LIN {X 0,Y 312.296,Z 514.961,A -85,B 0,C 180,E1 -15750.321,E2 -15750.321} C_VEL
LIN {X 0,Y 313.348,Z 507.271,A -85,B 0,C 180,E1 -15752.248,E2 -15752.248} C_VEL
LIN {X 0,Y 314.368,Z 497.665,A -85,B 0,C 180,E1 -15754.166,E2 -15754.166} C_VEL
LIN {X 0,Y 315.558,Z 488.778,A -85,B 0,C 180,E1 -15755.591,E2 -15755.591} C_VEL
LIN {X 0,Y 316.85,Z 477.877,A -85,B 0,C 180,E1 -15757.006,E2 -15757.006} C_VEL
LIN {X 0,Y 317.928,Z 465.494,A -85,B 0,C 180,E1 -15758.26,E2 -15758.26} C_VEL
LIN {X 0,Y 318.762,Z 453.367,A -85,B 0,C 180,E1 -15759.197,E2 -15759.197} C_VEL
LIN {X 0,Y 319.475,Z 440.605,A -85,B 0,C 180,E1 -15759.895,E2 -15759.895} C_VEL
LIN {X 0,Y 320.059,Z 427.037,A -85,B 0,C 180,E1 -15760.356,E2 -15760.356} C_VEL
LIN {X 0,Y 321.59,Z 354.256,A -85,B 0,C 180,E1 -15761.965,E2 -15761.965} C_VEL
LIN {X 0,Y 318.805,Z 337.841,A -85,B 0,C 180,E1 -15762.528,E2 -15762.528} C_VEL
LIN {X 0,Y 314.195,Z 324.041,A -85,B 0,C 180,E1 -15763.201,E2 -15763.201} C_VEL
LIN {X 0,Y 312.611,Z 316.546,A -85,B 0,C 180,E1 -15765.543,E2 -15765.543} C_VEL
LIN {X 0,Y 312.539,Z 316.555,A -85,B 0,C 180,E1 -15769.711,E2 -15769.711} C_VEL
LIN {X 0,Y 312.518,Z 316.554,A -85,B 0,C 180,E1 -15772.775,E2 -15772.775} C_VEL
LIN {X 0,Y 312.482,Z 316.56,A -85,B 0,C 180,E1 -15776.731,E2 -15776.731} C_VEL
LIN {X 0,Y 312.467,Z 316.56,A -85,B 0,C 180,E1 -15779.657,E2 -15779.657} C_VEL
LIN {X 0,Y 312.518,Z 316.553,A -85,B 0,C 180,E1 -15783.687,E2 -15783.687} C_VEL
LIN {X 0,Y 312.499,Z 316.556,A -85,B 0,C 180,E1 -15787.554,E2 -15787.554} C_VEL
LIN {X 0,Y 311.791,Z 316.649,A -85,B 0,C 180,E1 -15788.629,E2 -15788.629} C_VEL
LIN {X 0,Y 308.92,Z 317.003,A -85,B 0,C 180,E1 -15790.378,E2 -15790.378} C_VEL
LIN {X 0,Y 306.513,Z 317.302,A -85,B 0,C 180,E1 -15791.797,E2 -15791.797} C_VEL
LIN {X 0,Y 305.489,Z 317.434,A -85,B 0,C 180,E1 -15792.895,E2 -15792.895} C_VEL
LIN {X 0,Y 305.409,Z 317.438,A -85,B 0,C 180,E1 -15793.267,E2 -15793.267} C_VEL
LIN {X 0,Y 305.429,Z 317.435,A -85,B 0,C 180,E1 -15797.417,E2 -15797.417} C_VEL
LIN {X 0,Y 305.454,Z 317.434,A -85,B 0,C 180,E1 -15801.594,E2 -15801.594} C_VEL
LIN {X 0,Y 305.455,Z 317.431,A -85,B 0,C 180,E1 -15804.885,E2 -15804.885} C_VEL
LIN {X 0,Y 305.433,Z 317.435,A -85,B 0,C 180,E1 -15808.358,E2 -15808.358} C_VEL
LIN {X 0,Y 305.444,Z 317.437,A -85,B 0,C 180,E1 -15811.105,E2 -15811.105} C_VEL
LIN {X 0,Y 305.471,Z 317.426,A -85,B 0,C 180,E1 -15814.078,E2 -15814.078} C_VEL
LIN {X 0,Y 305.452,Z 317.434,A -85,B 0,C 180,E1 -15818.399,E2 -15818.399} C_VEL
LIN {X 0,Y 305.5,Z 317.428,A -85,B 0,C 180,E1 -15821.212,E2 -15821.212} C_VEL
LIN {X 0,Y 305.558,Z 317.415,A -85,B 0,C 180,E1 -15825.344,E2 -15825.344} C_VEL
LIN {X 0,Y 305.611,Z 317.414,A -85,B 0,C 180,E1 -15829.398,E2 -15829.398} C_VEL
LIN {X 0,Y 305.732,Z 317.402,A -85,B 0,C 180,E1 -15832.072,E2 -15832.072} C_VEL
LIN {X 0,Y 305.652,Z 317.403,A -85,B 0,C 180,E1 -15834.723,E2 -15834.723} C_VEL
LIN {X 0,Y 305.927,Z 317.376,A -85,B 0,C 180,E1 -15838.683,E2 -15838.683} C_VEL
LIN {X 0,Y 305.938,Z 317.372,A -85,B 0,C 180,E1 -15841.316,E2 -15841.316} C_VEL
LIN {X 0,Y 305.79,Z 317.391,A -85,B 0,C 180,E1 -15846.599,E2 -15846.599} C_VEL
LIN {X 0,Y 305.686,Z 317.405,A -85,B 0,C 180,E1 -15849.261,E2 -15849.261} C_VEL
LIN {X 0,Y 305.578,Z 317.417,A -85,B 0,C 180,E1 -15853.296,E2 -15853.296} C_VEL
LIN {X 0,Y 305.544,Z 317.417,A -85,B 0,C 180,E1 -15856.023,E2 -15856.023} C_VEL
LIN {X 0,Y 305.534,Z 317.425,A -85,B 0,C 180,E1 -15859.427,E2 -15859.427} C_VEL
LIN {X 0,Y 305.479,Z 317.433,A -85,B 0,C 180,E1 -15863.04,E2 -15863.04} C_VEL
LIN {X 0,Y 305.497,Z 317.427,A -85,B 0,C 180,E1 -15866.211,E2 -15866.211} C_VEL
LIN {X 0,Y 305.48,Z 317.432,A -85,B 0,C 180,E1 -15869.047,E2 -15869.047} C_VEL
LIN {X 0,Y 305.435,Z 317.435,A -85,B 0,C 180,E1 -15871.953,E2 -15871.953} C_VEL
LIN {X 0,Y 305.455,Z 317.435,A -85,B 0,C 180,E1 -15875.114,E2 -15875.114} C_VEL
LIN {X 0,Y 305.429,Z 317.436,A -85,B 0,C 180,E1 -15878.526,E2 -15878.526} C_VEL
LIN {X 0,Y 305.421,Z 317.438,A -85,B 0,C 180,E1 -15881.86,E2 -15881.86} C_VEL
LIN {X 0,Y 305.395,Z 317.444,A -85,B 0,C 180,E1 -15885.512,E2 -15885.512} C_VEL
LIN {X 0,Y 305.435,Z 317.439,A -85,B 0,C 180,E1 -15888.144,E2 -15888.144} C_VEL
LIN {X 0,Y 305.49,Z 317.432,A -85,B 0,C 180,E1 -15891.601,E2 -15891.601} C_VEL
LIN {X 0,Y 305.459,Z 317.434,A -85,B 0,C 180,E1 -15894.888,E2 -15894.888} C_VEL
LIN {X 0,Y 305.49,Z 317.525,A -85,B 0,C 180,E1 -15898.876,E2 -15898.876} C_VEL
LIN {X 0,Y 307.703,Z 328.091,A -85,B 0,C 180,E1 -15902.083,E2 -15902.083} C_VEL
LIN {X 0,Y 309.104,Z 336.061,A -85,B 0,C 180,E1 -15904.407,E2 -15904.407} C_VEL
LIN {X 0,Y 308.868,Z 340.002,A -85,B 0,C 180,E1 -15905.479,E2 -15905.479} C_VEL
LIN {X 0,Y 313.894,Z 375.423,A -85,B 0,C 180,E1 -15906.683,E2 -15906.683} C_VEL
LIN {X 0,Y 314.544,Z 381.837,A -85,B 0,C 180,E1 -15906.877,E2 -15906.877} C_VEL
LIN {X 0,Y 313.201,Z 448.115,A -85,B 0,C 180,E1 -15908.4,E2 -15908.4} C_VEL
LIN {X 0,Y 312.449,Z 461.495,A -85,B 0,C 180,E1 -15908.951,E2 -15908.951} C_VEL
LIN {X 0,Y 311.441,Z 473.727,A -85,B 0,C 180,E1 -15909.7,E2 -15909.7} C_VEL
LIN {X 0,Y 310.367,Z 485.256,A -85,B 0,C 180,E1 -15910.661,E2 -15910.661} C_VEL
LIN {X 0,Y 309.007,Z 497.067,A -85,B 0,C 180,E1 -15911.949,E2 -15911.949} C_VEL
LIN {X 0,Y 307.847,Z 507.337,A -85,B 0,C 180,E1 -15913.367,E2 -15913.367} C_VEL
LIN {X 0,Y 306.701,Z 517.217,A -85,B 0,C 180,E1 -15915.062,E2 -15915.062} C_VEL
LIN {X 0,Y 305.542,Z 526.379,A -85,B 0,C 180,E1 -15917.041,E2 -15917.041} C_VEL
LIN {X 0,Y 304.7,Z 533.755,A -85,B 0,C 180,E1 -15919.031,E2 -15919.031} C_VEL
LIN {X 0,Y 304.214,Z 538.742,A -85,B 0,C 180,E1 -15920.695,E2 -15920.695} C_VEL
LIN {X 0,Y 303.841,Z 543.574,A -85,B 0,C 180,E1 -15922.692,E2 -15922.692} C_VEL
LIN {X 0,Y 303.637,Z 547.267,A -85,B 0,C 180,E1 -15924.689,E2 -15924.689} C_VEL
LIN {X 0,Y 303.637,Z 549.173,A -85,B 0,C 180,E1 -15926.019,E2 -15926.019} C_VEL
LIN {X 0,Y 303.614,Z 550.618,A -85,B 0,C 180,E1 -15927.348,E2 -15927.348} C_VEL
LIN {X 0,Y 303.579,Z 551.634,A -85,B 0,C 180,E1 -15928.674,E2 -15928.674} C_VEL
LIN {X 0,Y 303.605,Z 552.26,A -85,B 0,C 180,E1 -15930.001,E2 -15930.001} C_VEL
LIN {X 0,Y 303.573,Z 552.497,A -85,B 0,C 180,E1 -15931.328,E2 -15931.328} C_VEL
LIN {X 0,Y 303.601,Z 552.318,A -85,B 0,C 180,E1 -15932.655,E2 -15932.655} C_VEL
LIN {X 0,Y 303.638,Z 550.75,A -85,B 0,C 180,E1 -15935.313,E2 -15935.313} C_VEL
LIN {X 0,Y 303.755,Z 549.383,A -85,B 0,C 180,E1 -15936.644,E2 -15936.644} C_VEL
LIN {X 0,Y 304.19,Z 546.513,A -85,B 0,C 180,E1 -15938.638,E2 -15938.638} C_VEL
LIN {X 0,Y 304.838,Z 542.633,A -85,B 0,C 180,E1 -15940.629,E2 -15940.629} C_VEL
LIN {X 0,Y 305.776,Z 537.648,A -85,B 0,C 180,E1 -15942.613,E2 -15942.613} C_VEL
LIN {X 0,Y 307.136,Z 531.405,A -85,B 0,C 180,E1 -15944.579,E2 -15944.579} C_VEL
LIN {X 0,Y 308.798,Z 523.623,A -85,B 0,C 180,E1 -15946.529,E2 -15946.529} C_VEL
LIN {X 0,Y 310.409,Z 514.991,A -85,B 0,C 180,E1 -15948.278,E2 -15948.278} C_VEL
LIN {X 0,Y 312.375,Z 505.012,A -85,B 0,C 180,E1 -15949.895,E2 -15949.895} C_VEL
LIN {X 0,Y 314.343,Z 494.038,A -85,B 0,C 180,E1 -15951.305,E2 -15951.305} C_VEL
LIN {X 0,Y 316.047,Z 483.306,A -85,B 0,C 180,E1 -15952.385,E2 -15952.385} C_VEL
LIN {X 0,Y 317.554,Z 471.518,A -85,B 0,C 180,E1 -15953.304,E2 -15953.304} C_VEL
LIN {X 0,Y 318.911,Z 458.823,A -85,B 0,C 180,E1 -15954.018,E2 -15954.018} C_VEL
LIN {X 0,Y 319.693,Z 446.646,A -85,B 0,C 180,E1 -15954.473,E2 -15954.473} C_VEL
LIN {X 0,Y 321.429,Z 382.108,A -85,B 0,C 180,E1 -15955.952,E2 -15955.952} C_VEL
LIN {X 0,Y 317.863,Z 362.317,A -85,B 0,C 180,E1 -15956.829,E2 -15956.829} C_VEL
LIN {X 0,Y 315.108,Z 349.801,A -85,B 0,C 180,E1 -15957.454,E2 -15957.454} C_VEL
LIN {X 0,Y 310.693,Z 339.327,A -85,B 0,C 180,E1 -15958.249,E2 -15958.249} C_VEL
LIN {X 0,Y 308.404,Z 329.1,A -85,B 0,C 180,E1 -15961.611,E2 -15961.611} C_VEL
LIN {X 0,Y 305.969,Z 319.3,A -85,B 0,C 180,E1 -15965.047,E2 -15965.047} C_VEL
LIN {X 0,Y 305.494,Z 317.433,A -85,B 0,C 180,E1 -15965.818,E2 -15965.818} C_VEL
LIN {X 0,Y 305.459,Z 317.436,A -85,B 0,C 180,E1 -15970.108,E2 -15970.108} C_VEL
LIN {X 0,Y 305.427,Z 317.437,A -85,B 0,C 180,E1 -15973.656,E2 -15973.656} C_VEL
LIN {X 0,Y 305.456,Z 317.436,A -85,B 0,C 180,E1 -15977.415,E2 -15977.415} C_VEL
LIN {X 0,Y 305.459,Z 317.434,A -85,B 0,C 180,E1 -15979.893,E2 -15979.893} C_VEL
LIN {X 0,Y 305.465,Z 317.433,A -85,B 0,C 180,E1 -15983.637,E2 -15983.637} C_VEL
LIN {X 0,Y 305.467,Z 317.435,A -85,B 0,C 180,E1 -15986.484,E2 -15986.484} C_VEL
LIN {X 0,Y 305.437,Z 317.438,A -85,B 0,C 180,E1 -15989.588,E2 -15989.588} C_VEL
LIN {X 0,Y 305.473,Z 317.43,A -85,B 0,C 180,E1 -15992.604,E2 -15992.604} C_VEL
LIN {X 0,Y 305.49,Z 317.426,A -85,B 0,C 180,E1 -15995.537,E2 -15995.537} C_VEL
LIN {X 0,Y 305.486,Z 317.428,A -85,B 0,C 180,E1 -15999.813,E2 -15999.813} C_VEL
LIN {X 0,Y 305.556,Z 317.418,A -85,B 0,C 180,E1 -16003.978,E2 -16003.978} C_VEL
LIN {X 0,Y 305.588,Z 317.412,A -85,B 0,C 180,E1 -16006.704,E2 -16006.704} C_VEL
LIN {X 0,Y 305.758,Z 317.389,A -85,B 0,C 180,E1 -16011.258,E2 -16011.258} C_VEL
LIN {X 0,Y 305.833,Z 317.382,A -85,B 0,C 180,E1 -16013.402,E2 -16013.402} C_VEL
LIN {X 0,Y 305.951,Z 317.368,A -85,B 0,C 180,E1 -16018.684,E2 -16018.684} C_VEL
LIN {X 0,Y 305.952,Z 317.364,A -85,B 0,C 180,E1 -16021.317,E2 -16021.317} C_VEL
LIN {X 0,Y 305.672,Z 317.399,A -85,B 0,C 180,E1 -16025.277,E2 -16025.277} C_VEL
LIN {X 0,Y 305.767,Z 317.396,A -85,B 0,C 180,E1 -16027.927,E2 -16027.927} C_VEL
LIN {X 0,Y 305.602,Z 317.417,A -85,B 0,C 180,E1 -16031.945,E2 -16031.945} C_VEL
LIN {X 0,Y 305.612,Z 317.418,A -85,B 0,C 180,E1 -16035.015,E2 -16035.015} C_VEL
LIN {X 0,Y 305.547,Z 317.423,A -85,B 0,C 180,E1 -16039.427,E2 -16039.427} C_VEL
LIN {X 0,Y 305.489,Z 317.431,A -85,B 0,C 180,E1 -16043.039,E2 -16043.039} C_VEL
LIN {X 0,Y 305.481,Z 317.428,A -85,B 0,C 180,E1 -16046.2,E2 -16046.2} C_VEL
LIN {X 0,Y 305.466,Z 317.428,A -85,B 0,C 180,E1 -16049.039,E2 -16049.039} C_VEL
LIN {X 0,Y 305.44,Z 317.432,A -85,B 0,C 180,E1 -16051.953,E2 -16051.953} C_VEL
LIN {X 0,Y 305.466,Z 317.43,A -85,B 0,C 180,E1 -16055.113,E2 -16055.113} C_VEL
LIN {X 0,Y 305.452,Z 317.437,A -85,B 0,C 180,E1 -16058.528,E2 -16058.528} C_VEL
LIN {X 0,Y 305.458,Z 317.436,A -85,B 0,C 180,E1 -16062.586,E2 -16062.586} C_VEL
LIN {X 0,Y 305.425,Z 317.441,A -85,B 0,C 180,E1 -16066.344,E2 -16066.344} C_VEL
LIN {X 0,Y 305.439,Z 317.538,A -85,B 0,C 180,E1 -16067.751,E2 -16067.751} C_VEL
LIN {X 0,Y 307.326,Z 324.783,A -85,B 0,C 180,E1 -16070.4,E2 -16070.4} C_VEL
LIN {X 0,Y 316.814,Z 344.367,A -85,B 0,C 180,E1 -16072.019,E2 -16072.019} C_VEL
LIN {X 0,Y 321.176,Z 354.703,A -85,B 0,C 180,E1 -16072.753,E2 -16072.753} C_VEL
LIN {X 0,Y 322.117,Z 358.964,A -85,B 0,C 180,E1 -16072.96,E2 -16072.96} C_VEL
LIN {X 0,Y 319.954,Z 432.294,A -85,B 0,C 180,E1 -16074.634,E2 -16074.634} C_VEL
LIN {X 0,Y 319.069,Z 445.156,A -85,B 0,C 180,E1 -16075.157,E2 -16075.157} C_VEL
LIN {X 0,Y 317.781,Z 458.257,A -85,B 0,C 180,E1 -16075.957,E2 -16075.957} C_VEL
LIN {X 0,Y 316.528,Z 468.963,A -85,B 0,C 180,E1 -16076.854,E2 -16076.854} C_VEL
LIN {X 0,Y 314.836,Z 480.903,A -85,B 0,C 180,E1 -16078.156,E2 -16078.156} C_VEL
LIN {X 0,Y 312.867,Z 491.723,A -85,B 0,C 180,E1 -16079.64,E2 -16079.64} C_VEL
LIN {X 0,Y 310.97,Z 501.278,A -85,B 0,C 180,E1 -16081.297,E2 -16081.297} C_VEL
LIN {X 0,Y 309.069,Z 510.472,A -85,B 0,C 180,E1 -16083.313,E2 -16083.313} C_VEL
LIN {X 0,Y 307.444,Z 517.806,A -85,B 0,C 180,E1 -16085.342,E2 -16085.342} C_VEL
LIN {X 0,Y 306.397,Z 522.72,A -85,B 0,C 180,E1 -16087.049,E2 -16087.049} C_VEL
LIN {X 0,Y 305.343,Z 527.44,A -85,B 0,C 180,E1 -16089.098,E2 -16089.098} C_VEL
LIN {X 0,Y 304.609,Z 530.992,A -85,B 0,C 180,E1 -16091.154,E2 -16091.154} C_VEL
LIN {X 0,Y 304.184,Z 532.749,A -85,B 0,C 180,E1 -16092.52,E2 -16092.52} C_VEL
LIN {X 0,Y 303.878,Z 534.072,A -85,B 0,C 180,E1 -16093.886,E2 -16093.886} C_VEL
LIN {X 0,Y 303.634,Z 535.444,A -85,B 0,C 180,E1 -16096.447,E2 -16096.447} C_VEL
LIN {X 0,Y 303.5,Z 535.534,A -85,B 0,C 180,E1 -16097.97,E2 -16097.97} C_VEL
LIN {X 0,Y 303.445,Z 534.477,A -85,B 0,C 180,E1 -16100.669,E2 -16100.669} C_VEL
LIN {X 0,Y 303.521,Z 533.321,A -85,B 0,C 180,E1 -16102.013,E2 -16102.013} C_VEL
LIN {X 0,Y 303.798,Z 530.629,A -85,B 0,C 180,E1 -16104.134,E2 -16104.134} C_VEL
LIN {X 0,Y 304.077,Z 527.294,A -85,B 0,C 180,E1 -16106.023,E2 -16106.023} C_VEL
LIN {X 0,Y 304.507,Z 522.685,A -85,B 0,C 180,E1 -16108.015,E2 -16108.015} C_VEL
LIN {X 0,Y 305.18,Z 515.732,A -85,B 0,C 180,E1 -16110.329,E2 -16110.329} C_VEL
LIN {X 0,Y 306.278,Z 508.187,A -85,B 0,C 180,E1 -16112.3,E2 -16112.3} C_VEL
LIN {X 0,Y 307.123,Z 500.516,A -85,B 0,C 180,E1 -16113.935,E2 -16113.935} C_VEL
LIN {X 0,Y 308.265,Z 491.148,A -85,B 0,C 180,E1 -16115.559,E2 -16115.559} C_VEL
LIN {X 0,Y 309.678,Z 480.703,A -85,B 0,C 180,E1 -16117.006,E2 -16117.006} C_VEL
LIN {X 0,Y 310.816,Z 469.157,A -85,B 0,C 180,E1 -16118.287,E2 -16118.287} C_VEL
LIN {X 0,Y 311.744,Z 456.945,A -85,B 0,C 180,E1 -16119.324,E2 -16119.324} C_VEL
LIN {X 0,Y 312.536,Z 444.098,A -85,B 0,C 180,E1 -16120.117,E2 -16120.117} C_VEL
LIN {X 0,Y 313.129,Z 431.64,A -85,B 0,C 180,E1 -16120.629,E2 -16120.629} C_VEL
LIN {X 0,Y 314.902,Z 355.1,A -85,B 0,C 180,E1 -16122.373,E2 -16122.373} C_VEL
LIN {X 0,Y 312.167,Z 339.4,A -85,B 0,C 180,E1 -16122.932,E2 -16122.932} C_VEL
LIN {X 0,Y 307.042,Z 324.32,A -85,B 0,C 180,E1 -16123.673,E2 -16123.673} C_VEL
LIN {X 0,Y 305.557,Z 317.426,A -85,B 0,C 180,E1 -16125.894,E2 -16125.894} C_VEL
LIN {X 0,Y 305.484,Z 317.435,A -85,B 0,C 180,E1 -16130.186,E2 -16130.186} C_VEL
LIN {X 0,Y 305.456,Z 317.437,A -85,B 0,C 180,E1 -16134.464,E2 -16134.464} C_VEL
LIN {X 0,Y 305.441,Z 317.435,A -85,B 0,C 180,E1 -16137.398,E2 -16137.398} C_VEL
LIN {X 0,Y 305.415,Z 317.442,A -85,B 0,C 180,E1 -16140.413,E2 -16140.413} C_VEL
LIN {X 0,Y 305.463,Z 317.433,A -85,B 0,C 180,E1 -16144.077,E2 -16144.077} C_VEL
LIN {X 0,Y 305.429,Z 317.436,A -85,B 0,C 180,E1 -16147.552,E2 -16147.552} C_VEL
LIN {X 0,Y 305.407,Z 317.438,A -85,B 0,C 180,E1 -16151.861,E2 -16151.861} C_VEL
LIN {X 0,Y 305.409,Z 317.438,A -85,B 0,C 180,E1 -16153.267,E2 -16153.267} C_VEL
LIN {X 0,Y 304.752,Z 317.523,A -85,B 0,C 180,E1 -16154.368,E2 -16154.368} C_VEL
LIN {X 0,Y 301.911,Z 317.881,A -85,B 0,C 180,E1 -16156.161,E2 -16156.161} C_VEL
LIN {X 0,Y 299.484,Z 318.183,A -85,B 0,C 180,E1 -16157.615,E2 -16157.615} C_VEL
LIN {X 0,Y 298.428,Z 318.311,A -85,B 0,C 180,E1 -16158.74,E2 -16158.74} C_VEL
LIN {X 0,Y 298.333,Z 318.32,A -85,B 0,C 180,E1 -16159.122,E2 -16159.122} C_VEL
LIN {X 0,Y 298.422,Z 318.31,A -85,B 0,C 180,E1 -16163.196,E2 -16163.196} C_VEL
LIN {X 0,Y 298.402,Z 318.31,A -85,B 0,C 180,E1 -16165.58,E2 -16165.58} C_VEL
LIN {X 0,Y 298.363,Z 318.317,A -85,B 0,C 180,E1 -16168.787,E2 -16168.787} C_VEL
LIN {X 0,Y 298.387,Z 318.312,A -85,B 0,C 180,E1 -16171.896,E2 -16171.896} C_VEL
LIN {X 0,Y 298.414,Z 318.304,A -85,B 0,C 180,E1 -16174.917,E2 -16174.917} C_VEL
LIN {X 0,Y 298.408,Z 318.313,A -85,B 0,C 180,E1 -16179.312,E2 -16179.312} C_VEL
LIN {X 0,Y 298.43,Z 318.307,A -85,B 0,C 180,E1 -16182.172,E2 -16182.172} C_VEL
LIN {X 0,Y 298.502,Z 318.291,A -85,B 0,C 180,E1 -16184.99,E2 -16184.99} C_VEL
LIN {X 0,Y 298.569,Z 318.29,A -85,B 0,C 180,E1 -16189.145,E2 -16189.145} C_VEL
LIN {X 0,Y 298.677,Z 318.281,A -85,B 0,C 180,E1 -16191.883,E2 -16191.883} C_VEL
LIN {X 0,Y 298.622,Z 318.278,A -85,B 0,C 180,E1 -16194.598,E2 -16194.598} C_VEL
LIN {X 0,Y 298.895,Z 318.252,A -85,B 0,C 180,E1 -16198.652,E2 -16198.652} C_VEL
LIN {X 0,Y 298.905,Z 318.249,A -85,B 0,C 180,E1 -16201.347,E2 -16201.347} C_VEL
LIN {X 0,Y 298.739,Z 318.27,A -85,B 0,C 180,E1 -16206.755,E2 -16206.755} C_VEL
LIN {X 0,Y 298.617,Z 318.284,A -85,B 0,C 180,E1 -16209.482,E2 -16209.482} C_VEL
LIN {X 0,Y 298.537,Z 318.292,A -85,B 0,C 180,E1 -16213.616,E2 -16213.616} C_VEL
LIN {X 0,Y 298.478,Z 318.298,A -85,B 0,C 180,E1 -16216.412,E2 -16216.412} C_VEL
LIN {X 0,Y 298.475,Z 318.303,A -85,B 0,C 180,E1 -16219.639,E2 -16219.639} C_VEL
LIN {X 0,Y 298.418,Z 318.31,A -85,B 0,C 180,E1 -16223.601,E2 -16223.601} C_VEL
LIN {X 0,Y 298.448,Z 318.307,A -85,B 0,C 180,E1 -16226.578,E2 -16226.578} C_VEL
LIN {X 0,Y 298.409,Z 318.313,A -85,B 0,C 180,E1 -16229.642,E2 -16229.642} C_VEL
LIN {X 0,Y 298.388,Z 318.313,A -85,B 0,C 180,E1 -16232.801,E2 -16232.801} C_VEL
LIN {X 0,Y 298.422,Z 318.309,A -85,B 0,C 180,E1 -16236.804,E2 -16236.804} C_VEL
LIN {X 0,Y 298.375,Z 318.315,A -85,B 0,C 180,E1 -16241.087,E2 -16241.087} C_VEL
LIN {X 0,Y 298.393,Z 318.311,A -85,B 0,C 180,E1 -16243.104,E2 -16243.104} C_VEL
LIN {X 0,Y 298.398,Z 318.312,A -85,B 0,C 180,E1 -16246.922,E2 -16246.922} C_VEL
LIN {X 0,Y 298.41,Z 318.311,A -85,B 0,C 180,E1 -16251.005,E2 -16251.005} C_VEL
LIN {X 0,Y 298.415,Z 318.315,A -85,B 0,C 180,E1 -16253.931,E2 -16253.931} C_VEL
LIN {X 0,Y 298.394,Z 318.319,A -85,B 0,C 180,E1 -16257.984,E2 -16257.984} C_VEL
LIN {X 0,Y 298.443,Z 318.417,A -85,B 0,C 180,E1 -16258.511,E2 -16258.511} C_VEL
LIN {X 0,Y 300.623,Z 328.791,A -85,B 0,C 180,E1 -16261.746,E2 -16261.746} C_VEL
LIN {X 0,Y 302.175,Z 338.091,A -85,B 0,C 180,E1 -16264.516,E2 -16264.516} C_VEL
LIN {X 0,Y 302.038,Z 339.794,A -85,B 0,C 180,E1 -16264.987,E2 -16264.987} C_VEL
LIN {X 0,Y 306.832,Z 373.458,A -85,B 0,C 180,E1 -16266.173,E2 -16266.173} C_VEL
LIN {X 0,Y 307.838,Z 382.335,A -85,B 0,C 180,E1 -16266.457,E2 -16266.457} C_VEL
LIN {X 0,Y 306.415,Z 448.885,A -85,B 0,C 180,E1 -16268.03,E2 -16268.03} C_VEL
LIN {X 0,Y 305.573,Z 462.705,A -85,B 0,C 180,E1 -16268.631,E2 -16268.631} C_VEL
LIN {X 0,Y 304.504,Z 475.613,A -85,B 0,C 180,E1 -16269.482,E2 -16269.482} C_VEL
LIN {X 0,Y 303.319,Z 487.411,A -85,B 0,C 180,E1 -16270.546,E2 -16270.546} C_VEL
LIN {X 0,Y 301.871,Z 498.77,A -85,B 0,C 180,E1 -16271.858,E2 -16271.858} C_VEL
LIN {X 0,Y 300.694,Z 509.168,A -85,B 0,C 180,E1 -16273.391,E2 -16273.391} C_VEL
LIN {X 0,Y 299.553,Z 518.223,A -85,B 0,C 180,E1 -16275.045,E2 -16275.045} C_VEL
LIN {X 0,Y 298.409,Z 527.186,A -85,B 0,C 180,E1 -16277.072,E2 -16277.072} C_VEL
LIN {X 0,Y 297.576,Z 534.367,A -85,B 0,C 180,E1 -16279.11,E2 -16279.11} C_VEL
LIN {X 0,Y 297.014,Z 540.079,A -85,B 0,C 180,E1 -16281.154,E2 -16281.154} C_VEL
LIN {X 0,Y 296.693,Z 544.567,A -85,B 0,C 180,E1 -16283.199,E2 -16283.199} C_VEL
LIN {X 0,Y 296.551,Z 546.928,A -85,B 0,C 180,E1 -16284.561,E2 -16284.561} C_VEL
LIN {X 0,Y 296.534,Z 548.857,A -85,B 0,C 180,E1 -16285.924,E2 -16285.924} C_VEL
LIN {X 0,Y 296.54,Z 550.346,A -85,B 0,C 180,E1 -16287.284,E2 -16287.284} C_VEL
LIN {X 0,Y 296.498,Z 551.383,A -85,B 0,C 180,E1 -16288.643,E2 -16288.643} C_VEL
LIN {X 0,Y 296.52,Z 552.03,A -85,B 0,C 180,E1 -16290.001,E2 -16290.001} C_VEL
LIN {X 0,Y 296.492,Z 552.288,A -85,B 0,C 180,E1 -16291.359,E2 -16291.359} C_VEL
LIN {X 0,Y 296.526,Z 552.148,A -85,B 0,C 180,E1 -16292.718,E2 -16292.718} C_VEL
LIN {X 0,Y 296.554,Z 550.625,A -85,B 0,C 180,E1 -16295.44,E2 -16295.44} C_VEL
LIN {X 0,Y 296.699,Z 549.281,A -85,B 0,C 180,E1 -16296.803,E2 -16296.803} C_VEL
LIN {X 0,Y 297.163,Z 546.456,A -85,B 0,C 180,E1 -16298.844,E2 -16298.844} C_VEL
LIN {X 0,Y 297.833,Z 542.625,A -85,B 0,C 180,E1 -16300.882,E2 -16300.882} C_VEL
LIN {X 0,Y 298.836,Z 537.691,A -85,B 0,C 180,E1 -16302.911,E2 -16302.911} C_VEL
LIN {X 0,Y 300.271,Z 531.505,A -85,B 0,C 180,E1 -16304.92,E2 -16304.92} C_VEL
LIN {X 0,Y 301.981,Z 523.823,A -85,B 0,C 180,E1 -16306.913,E2 -16306.913} C_VEL
LIN {X 0,Y 303.883,Z 514.218,A -85,B 0,C 180,E1 -16308.893,E2 -16308.893} C_VEL
LIN {X 0,Y 305.964,Z 504.32,A -85,B 0,C 180,E1 -16310.506,E2 -16310.506} C_VEL
LIN {X 0,Y 308.055,Z 493.18,A -85,B 0,C 180,E1 -16311.937,E2 -16311.937} C_VEL
LIN {X 0,Y 309.787,Z 482.295,A -85,B 0,C 180,E1 -16313.039,E2 -16313.039} C_VEL
LIN {X 0,Y 311.382,Z 470.284,A -85,B 0,C 180,E1 -16313.971,E2 -16313.971} C_VEL
LIN {X 0,Y 312.662,Z 457.946,A -85,B 0,C 180,E1 -16314.662,E2 -16314.662} C_VEL
LIN {X 0,Y 313.538,Z 445.216,A -85,B 0,C 180,E1 -16315.119,E2 -16315.119} C_VEL
LIN {X 0,Y 315.256,Z 383.061,A -85,B 0,C 180,E1 -16316.568,E2 -16316.568} C_VEL
LIN {X 0,Y 311.286,Z 361.291,A -85,B 0,C 180,E1 -16317.575,E2 -16317.575} C_VEL
LIN {X 0,Y 309.205,Z 352.32,A -85,B 0,C 180,E1 -16318.052,E2 -16318.052} C_VEL
LIN {X 0,Y 304.326,Z 341.341,A -85,B 0,C 180,E1 -16318.928,E2 -16318.928} C_VEL
LIN {X 0,Y 303.478,Z 339.127,A -85,B 0,C 180,E1 -16319.1,E2 -16319.1} C_VEL
LIN {X 0,Y 300.994,Z 328.318,A -85,B 0,C 180,E1 -16322.799,E2 -16322.799} C_VEL
LIN {X 0,Y 298.449,Z 318.312,A -85,B 0,C 180,E1 -16326.49,E2 -16326.49} C_VEL
LIN {X 0,Y 298.401,Z 318.313,A -85,B 0,C 180,E1 -16329.488,E2 -16329.488} C_VEL
LIN {X 0,Y 298.401,Z 318.314,A -85,B 0,C 180,E1 -16333.104,E2 -16333.104} C_VEL
LIN {X 0,Y 298.405,Z 318.315,A -85,B 0,C 180,E1 -16336.921,E2 -16336.921} C_VEL
LIN {X 0,Y 298.392,Z 318.311,A -85,B 0,C 180,E1 -16341.01,E2 -16341.01} C_VEL
LIN {X 0,Y 298.407,Z 318.312,A -85,B 0,C 180,E1 -16343.929,E2 -16343.929} C_VEL
LIN {X 0,Y 298.395,Z 318.311,A -85,B 0,C 180,E1 -16347.2,E2 -16347.2} C_VEL
LIN {X 0,Y 298.412,Z 318.311,A -85,B 0,C 180,E1 -16350.622,E2 -16350.622} C_VEL
LIN {X 0,Y 298.452,Z 318.303,A -85,B 0,C 180,E1 -16354.921,E2 -16354.921} C_VEL
LIN {X 0,Y 298.416,Z 318.31,A -85,B 0,C 180,E1 -16357.864,E2 -16357.864} C_VEL
LIN {X 0,Y 298.48,Z 318.302,A -85,B 0,C 180,E1 -16360.753,E2 -16360.753} C_VEL
LIN {X 0,Y 298.588,Z 318.288,A -85,B 0,C 180,E1 -16364.995,E2 -16364.995} C_VEL
LIN {X 0,Y 298.593,Z 318.285,A -85,B 0,C 180,E1 -16369.147,E2 -16369.147} C_VEL
LIN {X 0,Y 298.719,Z 318.264,A -85,B 0,C 180,E1 -16371.885,E2 -16371.885} C_VEL
LIN {X 0,Y 298.649,Z 318.276,A -85,B 0,C 180,E1 -16374.599,E2 -16374.599} C_VEL
LIN {X 0,Y 298.918,Z 318.244,A -85,B 0,C 180,E1 -16378.653,E2 -16378.653} C_VEL
LIN {X 0,Y 298.919,Z 318.24,A -85,B 0,C 180,E1 -16381.347,E2 -16381.347} C_VEL
LIN {X 0,Y 298.748,Z 318.27,A -85,B 0,C 180,E1 -16386.755,E2 -16386.755} C_VEL
LIN {X 0,Y 298.628,Z 318.276,A -85,B 0,C 180,E1 -16389.482,E2 -16389.482} C_VEL
LIN {X 0,Y 298.548,Z 318.287,A -85,B 0,C 180,E1 -16393.616,E2 -16393.616} C_VEL
LIN {X 0,Y 298.49,Z 318.302,A -85,B 0,C 180,E1 -16396.412,E2 -16396.412} C_VEL
LIN {X 0,Y 298.487,Z 318.302,A -85,B 0,C 180,E1 -16399.64,E2 -16399.64} C_VEL
LIN {X 0,Y 298.427,Z 318.308,A -85,B 0,C 180,E1 -16403.601,E2 -16403.601} C_VEL
LIN {X 0,Y 298.42,Z 318.309,A -85,B 0,C 180,E1 -16406.582,E2 -16406.582} C_VEL
LIN {X 0,Y 298.403,Z 318.313,A -85,B 0,C 180,E1 -16409.643,E2 -16409.643} C_VEL
LIN {X 0,Y 298.396,Z 318.313,A -85,B 0,C 180,E1 -16412.801,E2 -16412.801} C_VEL
LIN {X 0,Y 298.45,Z 318.307,A -85,B 0,C 180,E1 -16416.808,E2 -16416.808} C_VEL
LIN {X 0,Y 298.391,Z 318.318,A -85,B 0,C 180,E1 -16421.088,E2 -16421.088} C_VEL
LIN {X 0,Y 298.403,Z 318.316,A -85,B 0,C 180,E1 -16423.103,E2 -16423.103} C_VEL
LIN {X 0,Y 298.395,Z 318.392,A -85,B 0,C 180,E1 -16426.998,E2 -16426.998} C_VEL
LIN {X 0,Y 300.211,Z 325.283,A -85,B 0,C 180,E1 -16429.537,E2 -16429.537} C_VEL
LIN {X 0,Y 308.112,Z 340.972,A -85,B 0,C 180,E1 -16430.942,E2 -16430.942} C_VEL
LIN {X 0,Y 315.261,Z 357.011,A -85,B 0,C 180,E1 -16432.179,E2 -16432.179} C_VEL
LIN {X 0,Y 316.009,Z 361.29,A -85,B 0,C 180,E1 -16432.373,E2 -16432.373} C_VEL
LIN {X 0,Y 313.693,Z 433.005,A -85,B 0,C 180,E1 -16434.037,E2 -16434.037} C_VEL
LIN {X 0,Y 312.808,Z 445.372,A -85,B 0,C 180,E1 -16434.553,E2 -16434.553} C_VEL
LIN {X 0,Y 311.474,Z 458.463,A -85,B 0,C 180,E1 -16435.366,E2 -16435.366} C_VEL
LIN {X 0,Y 310.168,Z 469.162,A -85,B 0,C 180,E1 -16436.279,E2 -16436.279} C_VEL
LIN {X 0,Y 308.668,Z 479.473,A -85,B 0,C 180,E1 -16437.4,E2 -16437.4} C_VEL
LIN {X 0,Y 306.558,Z 490.814,A -85,B 0,C 180,E1 -16438.947,E2 -16438.947} C_VEL
LIN {X 0,Y 304.555,Z 500.621,A -85,B 0,C 180,E1 -16440.634,E2 -16440.634} C_VEL
LIN {X 0,Y 302.827,Z 508.579,A -85,B 0,C 180,E1 -16442.343,E2 -16442.343} C_VEL
LIN {X 0,Y 301.056,Z 516.298,A -85,B 0,C 180,E1 -16444.413,E2 -16444.413} C_VEL
LIN {X 0,Y 299.607,Z 522.452,A -85,B 0,C 180,E1 -16446.498,E2 -16446.498} C_VEL
LIN {X 0,Y 298.464,Z 527.274,A -85,B 0,C 180,E1 -16448.593,E2 -16448.593} C_VEL
LIN {X 0,Y 297.6,Z 531.15,A -85,B 0,C 180,E1 -16450.845,E2 -16450.845} C_VEL
LIN {X 0,Y 297.213,Z 532.765,A -85,B 0,C 180,E1 -16452.096,E2 -16452.096} C_VEL
LIN {X 0,Y 296.855,Z 534.13,A -85,B 0,C 180,E1 -16453.494,E2 -16453.494} C_VEL
LIN {X 0,Y 296.653,Z 535.087,A -85,B 0,C 180,E1 -16454.893,E2 -16454.893} C_VEL
LIN {X 0,Y 296.565,Z 535.65,A -85,B 0,C 180,E1 -16456.319,E2 -16456.319} C_VEL
LIN {X 0,Y 296.418,Z 535.756,A -85,B 0,C 180,E1 -16457.678,E2 -16457.678} C_VEL
LIN {X 0,Y 296.358,Z 534.779,A -85,B 0,C 180,E1 -16460.444,E2 -16460.444} C_VEL
LIN {X 0,Y 296.423,Z 533.698,A -85,B 0,C 180,E1 -16461.821,E2 -16461.821} C_VEL
LIN {X 0,Y 296.708,Z 530.802,A -85,B 0,C 180,E1 -16464.181,E2 -16464.181} C_VEL
LIN {X 0,Y 297.054,Z 526.427,A -85,B 0,C 180,E1 -16466.608,E2 -16466.608} C_VEL
LIN {X 0,Y 297.566,Z 521.528,A -85,B 0,C 180,E1 -16468.646,E2 -16468.646} C_VEL
LIN {X 0,Y 298.243,Z 515.372,A -85,B 0,C 180,E1 -16470.674,E2 -16470.674} C_VEL
LIN {X 0,Y 299.371,Z 507.685,A -85,B 0,C 180,E1 -16472.69,E2 -16472.69} C_VEL
LIN {X 0,Y 300.487,Z 498.078,A -85,B 0,C 180,E1 -16474.694,E2 -16474.694} C_VEL
LIN {X 0,Y 301.761,Z 489.19,A -85,B 0,C 180,E1 -16476.183,E2 -16476.183} C_VEL
LIN {X 0,Y 303.134,Z 478.292,A -85,B 0,C 180,E1 -16477.66,E2 -16477.66} C_VEL
LIN {X 0,Y 304.296,Z 465.91,A -85,B 0,C 180,E1 -16478.968,E2 -16478.968} C_VEL
LIN {X 0,Y 305.193,Z 453.785,A -85,B 0,C 180,E1 -16479.944,E2 -16479.944} C_VEL
LIN {X 0,Y 305.958,Z 441.034,A -85,B 0,C 180,E1 -16480.672,E2 -16480.672} C_VEL
LIN {X 0,Y 306.585,Z 427.482,A -85,B 0,C 180,E1 -16481.151,E2 -16481.151} C_VEL
LIN {X 0,Y 308.261,Z 356.338,A -85,B 0,C 180,E1 -16482.786,E2 -16482.786} C_VEL
LIN {X 0,Y 305.757,Z 341.572,A -85,B 0,C 180,E1 -16483.322,E2 -16483.322} C_VEL
LIN {X 0,Y 299.86,Z 324.543,A -85,B 0,C 180,E1 -16484.187,E2 -16484.187} C_VEL
LIN {X 0,Y 298.486,Z 318.307,A -85,B 0,C 180,E1 -16486.261,E2 -16486.261} C_VEL
LIN {X 0,Y 298.447,Z 318.311,A -85,B 0,C 180,E1 -16489.618,E2 -16489.618} C_VEL
LIN {X 0,Y 298.409,Z 318.312,A -85,B 0,C 180,E1 -16493.6,E2 -16493.6} C_VEL
LIN {X 0,Y 298.401,Z 318.315,A -85,B 0,C 180,E1 -16496.582,E2 -16496.582} C_VEL
LIN {X 0,Y 298.356,Z 318.318,A -85,B 0,C 180,E1 -16499.647,E2 -16499.647} C_VEL
LIN {X 0,Y 298.391,Z 318.315,A -85,B 0,C 180,E1 -16502.799,E2 -16502.799} C_VEL
LIN {X 0,Y 298.438,Z 318.311,A -85,B 0,C 180,E1 -16506.805,E2 -16506.805} C_VEL
LIN {X 0,Y 298.344,Z 318.32,A -85,B 0,C 180,E1 -16511.077,E2 -16511.077} C_VEL
LIN {X 0,Y 298.351,Z 318.32,A -85,B 0,C 180,E1 -16515.034,E2 -16515.034} C_VEL
LIN {X 0,Y 298.343,Z 318.32,A -85,B 0,C 180,E1 -16518.92,E2 -16518.92} C_VEL
LIN {X 0,Y 298.333,Z 318.32,A -85,B 0,C 180,E1 -16519.122,E2 -16519.122} C_VEL
LIN {X 0,Y 297.665,Z 318.404,A -85,B 0,C 180,E1 -16520.25,E2 -16520.25} C_VEL
LIN {X 0,Y 294.884,Z 318.75,A -85,B 0,C 180,E1 -16522.089,E2 -16522.089} C_VEL
LIN {X 0,Y 292.514,Z 319.048,A -85,B 0,C 180,E1 -16523.58,E2 -16523.58} C_VEL
LIN {X 0,Y 291.464,Z 319.175,A -85,B 0,C 180,E1 -16524.734,E2 -16524.734} C_VEL
LIN {X 0,Y 291.36,Z 319.186,A -85,B 0,C 180,E1 -16525.124,E2 -16525.124} C_VEL
LIN {X 0,Y 291.358,Z 319.189,A -85,B 0,C 180,E1 -16527.948,E2 -16527.948} C_VEL
LIN {X 0,Y 291.307,Z 319.198,A -85,B 0,C 180,E1 -16531.15,E2 -16531.15} C_VEL
LIN {X 0,Y 291.339,Z 319.184,A -85,B 0,C 180,E1 -16534.264,E2 -16534.264} C_VEL
LIN {X 0,Y 291.343,Z 319.191,A -85,B 0,C 180,E1 -16537.296,E2 -16537.296} C_VEL
LIN {X 0,Y 291.378,Z 319.187,A -85,B 0,C 180,E1 -16540.264,E2 -16540.264} C_VEL
LIN {X 0,Y 291.444,Z 319.17,A -85,B 0,C 180,E1 -16544.698,E2 -16544.698} C_VEL
LIN {X 0,Y 291.513,Z 319.169,A -85,B 0,C 180,E1 -16548.879,E2 -16548.879} C_VEL
LIN {X 0,Y 291.623,Z 319.158,A -85,B 0,C 180,E1 -16551.686,E2 -16551.686} C_VEL
LIN {X 0,Y 291.591,Z 319.154,A -85,B 0,C 180,E1 -16554.467,E2 -16554.467} C_VEL
LIN {X 0,Y 291.862,Z 319.128,A -85,B 0,C 180,E1 -16558.62,E2 -16558.62} C_VEL
LIN {X 0,Y 291.871,Z 319.125,A -85,B 0,C 180,E1 -16561.38,E2 -16561.38} C_VEL
LIN {X 0,Y 291.691,Z 319.146,A -85,B 0,C 180,E1 -16566.919,E2 -16566.919} C_VEL
LIN {X 0,Y 291.56,Z 319.163,A -85,B 0,C 180,E1 -16569.714,E2 -16569.714} C_VEL
LIN {X 0,Y 291.507,Z 319.168,A -85,B 0,C 180,E1 -16573.951,E2 -16573.951} C_VEL
LIN {X 0,Y 291.425,Z 319.179,A -85,B 0,C 180,E1 -16576.821,E2 -16576.821} C_VEL
LIN {X 0,Y 291.416,Z 319.182,A -85,B 0,C 180,E1 -16579.86,E2 -16579.86} C_VEL
LIN {X 0,Y 291.365,Z 319.187,A -85,B 0,C 180,E1 -16584.208,E2 -16584.208} C_VEL
LIN {X 0,Y 291.395,Z 319.187,A -85,B 0,C 180,E1 -16587.274,E2 -16587.274} C_VEL
LIN {X 0,Y 291.327,Z 319.193,A -85,B 0,C 180,E1 -16590.438,E2 -16590.438} C_VEL
LIN {X 0,Y 291.338,Z 319.194,A -85,B 0,C 180,E1 -16593.699,E2 -16593.699} C_VEL
LIN {X 0,Y 291.353,Z 319.192,A -85,B 0,C 180,E1 -16597.25,E2 -16597.25} C_VEL
LIN {X 0,Y 291.322,Z 319.192,A -85,B 0,C 180,E1 -16600.644,E2 -16600.644} C_VEL
LIN {X 0,Y 291.285,Z 319.199,A -85,B 0,C 180,E1 -16604.403,E2 -16604.403} C_VEL
LIN {X 0,Y 291.321,Z 319.196,A -85,B 0,C 180,E1 -16608.406,E2 -16608.406} C_VEL
LIN {X 0,Y 291.359,Z 319.19,A -85,B 0,C 180,E1 -16611.161,E2 -16611.161} C_VEL
LIN {X 0,Y 291.358,Z 319.192,A -85,B 0,C 180,E1 -16614.627,E2 -16614.627} C_VEL
LIN {X 0,Y 291.374,Z 319.24,A -85,B 0,C 180,E1 -16618.105,E2 -16618.105} C_VEL
LIN {X 0,Y 293.286,Z 328.16,A -85,B 0,C 180,E1 -16620.973,E2 -16620.973} C_VEL
LIN {X 0,Y 295.157,Z 338.808,A -85,B 0,C 180,E1 -16624.245,E2 -16624.245} C_VEL
LIN {X 0,Y 295.192,Z 339.601,A -85,B 0,C 180,E1 -16624.477,E2 -16624.477} C_VEL
LIN {X 0,Y 299.493,Z 369.307,A -85,B 0,C 180,E1 -16625.563,E2 -16625.563} C_VEL
LIN {X 0,Y 301.149,Z 382.977,A -85,B 0,C 180,E1 -16626.022,E2 -16626.022} C_VEL
LIN {X 0,Y 299.7,Z 448.507,A -85,B 0,C 180,E1 -16627.602,E2 -16627.602} C_VEL
LIN {X 0,Y 298.827,Z 462.384,A -85,B 0,C 180,E1 -16628.215,E2 -16628.215} C_VEL
LIN {X 0,Y 297.801,Z 474.289,A -85,B 0,C 180,E1 -16628.998,E2 -16628.998} C_VEL
LIN {X 0,Y 296.539,Z 486.343,A -85,B 0,C 180,E1 -16630.082,E2 -16630.082} C_VEL
LIN {X 0,Y 295.11,Z 497.871,A -85,B 0,C 180,E1 -16631.428,E2 -16631.428} C_VEL
LIN {X 0,Y 293.798,Z 508.657,A -85,B 0,C 180,E1 -16633.03,E2 -16633.03} C_VEL
LIN {X 0,Y 292.679,Z 517.584,A -85,B 0,C 180,E1 -16634.685,E2 -16634.685} C_VEL
LIN {X 0,Y 291.455,Z 526.618,A -85,B 0,C 180,E1 -16636.758,E2 -16636.758} C_VEL
LIN {X 0,Y 290.556,Z 533.88,A -85,B 0,C 180,E1 -16638.844,E2 -16638.844} C_VEL
LIN {X 0,Y 289.984,Z 539.662,A -85,B 0,C 180,E1 -16640.937,E2 -16640.937} C_VEL
LIN {X 0,Y 289.635,Z 544.201,A -85,B 0,C 180,E1 -16643.033,E2 -16643.033} C_VEL
LIN {X 0,Y 289.478,Z 546.705,A -85,B 0,C 180,E1 -16644.506,E2 -16644.506} C_VEL
LIN {X 0,Y 289.467,Z 550.065,A -85,B 0,C 180,E1 -16647.218,E2 -16647.218} C_VEL
LIN {X 0,Y 289.42,Z 551.131,A -85,B 0,C 180,E1 -16648.61,E2 -16648.61} C_VEL
LIN {X 0,Y 289.437,Z 551.8,A -85,B 0,C 180,E1 -16650.001,E2 -16650.001} C_VEL
LIN {X 0,Y 289.413,Z 552.078,A -85,B 0,C 180,E1 -16651.392,E2 -16651.392} C_VEL
LIN {X 0,Y 289.43,Z 551.971,A -85,B 0,C 180,E1 -16652.785,E2 -16652.785} C_VEL
LIN {X 0,Y 289.48,Z 550.501,A -85,B 0,C 180,E1 -16655.574,E2 -16655.574} C_VEL
LIN {X 0,Y 289.927,Z 547.457,A -85,B 0,C 180,E1 -16658.364,E2 -16658.364} C_VEL
LIN {X 0,Y 290.559,Z 544.015,A -85,B 0,C 180,E1 -16660.453,E2 -16660.453} C_VEL
LIN {X 0,Y 291.488,Z 539.513,A -85,B 0,C 180,E1 -16662.534,E2 -16662.534} C_VEL
LIN {X 0,Y 293.125,Z 532.721,A -85,B 0,C 180,E1 -16664.937,E2 -16664.937} C_VEL
LIN {X 0,Y 294.908,Z 525.372,A -85,B 0,C 180,E1 -16666.973,E2 -16666.973} C_VEL
LIN {X 0,Y 296.791,Z 516.442,A -85,B 0,C 180,E1 -16668.967,E2 -16668.967} C_VEL
LIN {X 0,Y 298.859,Z 506.84,A -85,B 0,C 180,E1 -16670.656,E2 -16670.656} C_VEL
LIN {X 0,Y 300.973,Z 496.399,A -85,B 0,C 180,E1 -16672.12,E2 -16672.12} C_VEL
LIN {X 0,Y 303.023,Z 484.804,A -85,B 0,C 180,E1 -16673.403,E2 -16673.403} C_VEL
LIN {X 0,Y 304.655,Z 473.589,A -85,B 0,C 180,E1 -16674.354,E2 -16674.354} C_VEL
LIN {X 0,Y 306.227,Z 460.254,A -85,B 0,C 180,E1 -16675.17,E2 -16675.17} C_VEL
LIN {X 0,Y 307.269,Z 446.839,A -85,B 0,C 180,E1 -16675.714,E2 -16675.714} C_VEL
LIN {X 0,Y 309.158,Z 384.274,A -85,B 0,C 180,E1 -16677.2,E2 -16677.2} C_VEL
LIN {X 0,Y 304.963,Z 361.053,A -85,B 0,C 180,E1 -16678.309,E2 -16678.309} C_VEL
LIN {X 0,Y 303.338,Z 354.788,A -85,B 0,C 180,E1 -16678.675,E2 -16678.675} C_VEL
LIN {X 0,Y 298.085,Z 342.904,A -85,B 0,C 180,E1 -16679.66,E2 -16679.66} C_VEL
LIN {X 0,Y 296.163,Z 338.801,A -85,B 0,C 180,E1 -16680.054,E2 -16680.054} C_VEL
LIN {X 0,Y 294.034,Z 329.501,A -85,B 0,C 180,E1 -16683.35,E2 -16683.35} C_VEL
LIN {X 0,Y 291.855,Z 320.959,A -85,B 0,C 180,E1 -16686.584,E2 -16686.584} C_VEL
LIN {X 0,Y 291.38,Z 319.19,A -85,B 0,C 180,E1 -16687.348,E2 -16687.348} C_VEL
LIN {X 0,Y 291.333,Z 319.196,A -85,B 0,C 180,E1 -16690.643,E2 -16690.643} C_VEL
LIN {X 0,Y 291.292,Z 319.2,A -85,B 0,C 180,E1 -16694.402,E2 -16694.402} C_VEL
LIN {X 0,Y 291.327,Z 319.193,A -85,B 0,C 180,E1 -16698.405,E2 -16698.405} C_VEL
LIN {X 0,Y 291.341,Z 319.189,A -85,B 0,C 180,E1 -16701.156,E2 -16701.156} C_VEL
LIN {X 0,Y 291.357,Z 319.187,A -85,B 0,C 180,E1 -16704.626,E2 -16704.626} C_VEL
LIN {X 0,Y 291.368,Z 319.183,A -85,B 0,C 180,E1 -16707.95,E2 -16707.95} C_VEL
LIN {X 0,Y 291.356,Z 319.186,A -85,B 0,C 180,E1 -16711.156,E2 -16711.156} C_VEL
LIN {X 0,Y 291.378,Z 319.188,A -85,B 0,C 180,E1 -16714.268,E2 -16714.268} C_VEL
LIN {X 0,Y 291.373,Z 319.192,A -85,B 0,C 180,E1 -16717.299,E2 -16717.299} C_VEL
LIN {X 0,Y 291.408,Z 319.182,A -85,B 0,C 180,E1 -16720.267,E2 -16720.267} C_VEL
LIN {X 0,Y 291.5,Z 319.169,A -85,B 0,C 180,E1 -16724.665,E2 -16724.665} C_VEL
LIN {X 0,Y 291.537,Z 319.163,A -85,B 0,C 180,E1 -16728.881,E2 -16728.881} C_VEL
LIN {X 0,Y 291.669,Z 319.141,A -85,B 0,C 180,E1 -16731.688,E2 -16731.688} C_VEL
LIN {X 0,Y 291.619,Z 319.153,A -85,B 0,C 180,E1 -16734.468,E2 -16734.468} C_VEL
LIN {X 0,Y 291.884,Z 319.121,A -85,B 0,C 180,E1 -16738.621,E2 -16738.621} C_VEL
LIN {X 0,Y 291.886,Z 319.116,A -85,B 0,C 180,E1 -16741.38,E2 -16741.38} C_VEL
LIN {X 0,Y 291.7,Z 319.147,A -85,B 0,C 180,E1 -16746.919,E2 -16746.919} C_VEL
LIN {X 0,Y 291.571,Z 319.156,A -85,B 0,C 180,E1 -16749.714,E2 -16749.714} C_VEL
LIN {X 0,Y 291.518,Z 319.163,A -85,B 0,C 180,E1 -16753.951,E2 -16753.951} C_VEL
LIN {X 0,Y 291.444,Z 319.173,A -85,B 0,C 180,E1 -16758.27,E2 -16758.27} C_VEL
LIN {X 0,Y 291.362,Z 319.183,A -85,B 0,C 180,E1 -16761.212,E2 -16761.212} C_VEL
LIN {X 0,Y 291.37,Z 319.187,A -85,B 0,C 180,E1 -16764.208,E2 -16764.208} C_VEL
LIN {X 0,Y 291.365,Z 319.188,A -85,B 0,C 180,E1 -16767.278,E2 -16767.278} C_VEL
LIN {X 0,Y 291.325,Z 319.194,A -85,B 0,C 180,E1 -16770.439,E2 -16770.439} C_VEL
LIN {X 0,Y 291.347,Z 319.191,A -85,B 0,C 180,E1 -16773.699,E2 -16773.699} C_VEL
LIN {X 0,Y 291.379,Z 319.186,A -85,B 0,C 180,E1 -16777.254,E2 -16777.254} C_VEL
LIN {X 0,Y 291.336,Z 319.195,A -85,B 0,C 180,E1 -16780.643,E2 -16780.643} C_VEL
LIN {X 0,Y 291.294,Z 319.199,A -85,B 0,C 180,E1 -16784.402,E2 -16784.402} C_VEL
LIN {X 0,Y 291.332,Z 319.406,A -85,B 0,C 180,E1 -16786.251,E2 -16786.251} C_VEL
LIN {X 0,Y 292.905,Z 325.297,A -85,B 0,C 180,E1 -16788.574,E2 -16788.574} C_VEL
LIN {X 0,Y 301.461,Z 341.936,A -85,B 0,C 180,E1 -16790.164,E2 -16790.164} C_VEL
LIN {X 0,Y 308.435,Z 357.264,A -85,B 0,C 180,E1 -16791.42,E2 -16791.42} C_VEL
LIN {X 0,Y 309.702,Z 360.793,A -85,B 0,C 180,E1 -16791.66,E2 -16791.66} C_VEL
LIN {X 0,Y 309.763,Z 366.14,A -85,B 0,C 180,E1 -16791.81,E2 -16791.81} C_VEL
LIN {X 0,Y 307.506,Z 433.178,A -85,B 0,C 180,E1 -16793.395,E2 -16793.395} C_VEL
LIN {X 0,Y 306.592,Z 445.631,A -85,B 0,C 180,E1 -16793.925,E2 -16793.925} C_VEL
LIN {X 0,Y 305.205,Z 458.705,A -85,B 0,C 180,E1 -16794.751,E2 -16794.751} C_VEL
LIN {X 0,Y 303.836,Z 469.391,A -85,B 0,C 180,E1 -16795.679,E2 -16795.679} C_VEL
LIN {X 0,Y 302.238,Z 479.836,A -85,B 0,C 180,E1 -16796.838,E2 -16796.838} C_VEL
LIN {X 0,Y 300.065,Z 491.028,A -85,B 0,C 180,E1 -16798.394,E2 -16798.394} C_VEL
LIN {X 0,Y 298.158,Z 499.916,A -85,B 0,C 180,E1 -16799.94,E2 -16799.94} C_VEL
LIN {X 0,Y 296.333,Z 508.053,A -85,B 0,C 180,E1 -16801.683,E2 -16801.683} C_VEL
LIN {X 0,Y 294.408,Z 515.922,A -85,B 0,C 180,E1 -16803.792,E2 -16803.792} C_VEL
LIN {X 0,Y 292.87,Z 522.185,A -85,B 0,C 180,E1 -16805.923,E2 -16805.923} C_VEL
LIN {X 0,Y 291.62,Z 527.107,A -85,B 0,C 180,E1 -16808.065,E2 -16808.065} C_VEL
LIN {X 0,Y 290.585,Z 531.429,A -85,B 0,C 180,E1 -16810.605,E2 -16810.605} C_VEL
LIN {X 0,Y 289.846,Z 534.188,A -85,B 0,C 180,E1 -16813.083,E2 -16813.083} C_VEL
LIN {X 0,Y 289.604,Z 535.187,A -85,B 0,C 180,E1 -16814.517,E2 -16814.517} C_VEL
LIN {X 0,Y 289.469,Z 535.862,A -85,B 0,C 180,E1 -16816.208,E2 -16816.208} C_VEL
LIN {X 0,Y 289.272,Z 535.724,A -85,B 0,C 180,E1 -16818.792,E2 -16818.792} C_VEL
LIN {X 0,Y 289.263,Z 535.081,A -85,B 0,C 180,E1 -16820.207,E2 -16820.207} C_VEL
LIN {X 0,Y 289.31,Z 534.047,A -85,B 0,C 180,E1 -16821.618,E2 -16821.618} C_VEL
LIN {X 0,Y 289.621,Z 530.984,A -85,B 0,C 180,E1 -16824.224,E2 -16824.224} C_VEL
LIN {X 0,Y 289.959,Z 526.982,A -85,B 0,C 180,E1 -16826.525,E2 -16826.525} C_VEL
LIN {X 0,Y 290.474,Z 522.179,A -85,B 0,C 180,E1 -16828.613,E2 -16828.613} C_VEL
LIN {X 0,Y 291.126,Z 516.131,A -85,B 0,C 180,E1 -16830.691,E2 -16830.691} C_VEL
LIN {X 0,Y 292.276,Z 508.588,A -85,B 0,C 180,E1 -16832.755,E2 -16832.755} C_VEL
LIN {X 0,Y 293.217,Z 500.915,A -85,B 0,C 180,E1 -16834.467,E2 -16834.467} C_VEL
LIN {X 0,Y 294.448,Z 491.548,A -85,B 0,C 180,E1 -16836.165,E2 -16836.165} C_VEL
LIN {X 0,Y 295.964,Z 481.1,A -85,B 0,C 180,E1 -16837.675,E2 -16837.675} C_VEL
LIN {X 0,Y 297.185,Z 469.555,A -85,B 0,C 180,E1 -16839.013,E2 -16839.013} C_VEL
LIN {X 0,Y 298.186,Z 457.345,A -85,B 0,C 180,E1 -16840.095,E2 -16840.095} C_VEL
LIN {X 0,Y 299.038,Z 444.501,A -85,B 0,C 180,E1 -16840.922,E2 -16840.922} C_VEL
LIN {X 0,Y 299.676,Z 432.047,A -85,B 0,C 180,E1 -16841.455,E2 -16841.455} C_VEL
LIN {X 0,Y 301.591,Z 357.276,A -85,B 0,C 180,E1 -16843.226,E2 -16843.226} C_VEL
LIN {X 0,Y 299.312,Z 343.654,A -85,B 0,C 180,E1 -16843.734,E2 -16843.734} C_VEL
LIN {X 0,Y 292.66,Z 324.694,A -85,B 0,C 180,E1 -16844.752,E2 -16844.752} C_VEL
LIN {X 0,Y 291.431,Z 319.185,A -85,B 0,C 180,E1 -16846.647,E2 -16846.647} C_VEL
LIN {X 0,Y 291.392,Z 319.191,A -85,B 0,C 180,E1 -16849.841,E2 -16849.841} C_VEL
LIN {X 0,Y 291.346,Z 319.196,A -85,B 0,C 180,E1 -16854.209,E2 -16854.209} C_VEL
LIN {X 0,Y 291.328,Z 319.193,A -85,B 0,C 180,E1 -16857.28,E2 -16857.28} C_VEL
LIN {X 0,Y 291.3,Z 319.2,A -85,B 0,C 180,E1 -16860.44,E2 -16860.44} C_VEL
LIN {X 0,Y 291.342,Z 319.191,A -85,B 0,C 180,E1 -16863.697,E2 -16863.697} C_VEL
LIN {X 0,Y 291.365,Z 319.189,A -85,B 0,C 180,E1 -16867.25,E2 -16867.25} C_VEL
LIN {X 0,Y 291.296,Z 319.198,A -85,B 0,C 180,E1 -16870.647,E2 -16870.647} C_VEL
LIN {X 0,Y 291.278,Z 319.201,A -85,B 0,C 180,E1 -16874.402,E2 -16874.402} C_VEL
LIN {X 0,Y 291.29,Z 319.195,A -85,B 0,C 180,E1 -16878.41,E2 -16878.41} C_VEL
LIN {X 0,Y 291.329,Z 319.196,A -85,B 0,C 180,E1 -16881.154,E2 -16881.154} C_VEL
LIN {X 0,Y 291.349,Z 319.186,A -85,B 0,C 180,E1 -16884.624,E2 -16884.624} C_VEL
LIN {X 0,Y 291.36,Z 319.186,A -85,B 0,C 180,E1 -16885.124,E2 -16885.124} C_VEL
LIN {X 0,Y 290.643,Z 319.274,A -85,B 0,C 180,E1 -16886.278,E2 -16886.278} C_VEL
LIN {X 0,Y 287.776,Z 319.634,A -85,B 0,C 180,E1 -16888.156,E2 -16888.156} C_VEL
LIN {X 0,Y 285.371,Z 319.937,A -85,B 0,C 180,E1 -16889.681,E2 -16889.681} C_VEL
LIN {X 0,Y 284.335,Z 320.064,A -85,B 0,C 180,E1 -16890.862,E2 -16890.862} C_VEL
LIN {X 0,Y 284.246,Z 320.069,A -85,B 0,C 180,E1 -16891.262,E2 -16891.262} C_VEL
LIN {X 0,Y 284.281,Z 320.064,A -85,B 0,C 180,E1 -16895.148,E2 -16895.148} C_VEL
LIN {X 0,Y 284.291,Z 320.07,A -85,B 0,C 180,E1 -16898.234,E2 -16898.234} C_VEL
LIN {X 0,Y 284.309,Z 320.068,A -85,B 0,C 180,E1 -16901.255,E2 -16901.255} C_VEL
LIN {X 0,Y 284.412,Z 320.045,A -85,B 0,C 180,E1 -16904.512,E2 -16904.512} C_VEL
LIN {X 0,Y 284.444,Z 320.051,A -85,B 0,C 180,E1 -16908.599,E2 -16908.599} C_VEL
LIN {X 0,Y 284.573,Z 320.035,A -85,B 0,C 180,E1 -16911.478,E2 -16911.478} C_VEL
LIN {X 0,Y 284.561,Z 320.029,A -85,B 0,C 180,E1 -16914.33,E2 -16914.33} C_VEL
LIN {X 0,Y 284.83,Z 320.004,A -85,B 0,C 180,E1 -16918.586,E2 -16918.586} C_VEL
LIN {X 0,Y 284.837,Z 320.001,A -85,B 0,C 180,E1 -16921.414,E2 -16921.414} C_VEL
LIN {X 0,Y 284.646,Z 320.022,A -85,B 0,C 180,E1 -16927.091,E2 -16927.091} C_VEL
LIN {X 0,Y 284.506,Z 320.043,A -85,B 0,C 180,E1 -16929.957,E2 -16929.957} C_VEL
LIN {X 0,Y 284.455,Z 320.047,A -85,B 0,C 180,E1 -16934.304,E2 -16934.304} C_VEL
LIN {X 0,Y 284.355,Z 320.063,A -85,B 0,C 180,E1 -16938.742,E2 -16938.742} C_VEL
LIN {X 0,Y 284.307,Z 320.067,A -85,B 0,C 180,E1 -16941.765,E2 -16941.765} C_VEL
LIN {X 0,Y 284.316,Z 320.068,A -85,B 0,C 180,E1 -16944.849,E2 -16944.849} C_VEL
LIN {X 0,Y 284.309,Z 320.065,A -85,B 0,C 180,E1 -16948.013,E2 -16948.013} C_VEL
LIN {X 0,Y 284.287,Z 320.075,A -85,B 0,C 180,E1 -16951.275,E2 -16951.275} C_VEL
LIN {X 0,Y 284.33,Z 320.069,A -85,B 0,C 180,E1 -16955.347,E2 -16955.347} C_VEL
LIN {X 0,Y 284.296,Z 320.07,A -85,B 0,C 180,E1 -16958.171,E2 -16958.171} C_VEL
LIN {X 0,Y 284.246,Z 320.073,A -85,B 0,C 180,E1 -16962.121,E2 -16962.121} C_VEL
LIN {X 0,Y 284.251,Z 320.077,A -85,B 0,C 180,E1 -16966.19,E2 -16966.19} C_VEL
LIN {X 0,Y 284.303,Z 320.072,A -85,B 0,C 180,E1 -16970.025,E2 -16970.025} C_VEL
LIN {X 0,Y 284.331,Z 320.067,A -85,B 0,C 180,E1 -16973.616,E2 -16973.616} C_VEL
LIN {X 0,Y 284.335,Z 320.194,A -85,B 0,C 180,E1 -16977.724,E2 -16977.724} C_VEL
LIN {X 0,Y 286.438,Z 330.002,A -85,B 0,C 180,E1 -16980.96,E2 -16980.96} C_VEL
LIN {X 0,Y 288.129,Z 339.437,A -85,B 0,C 180,E1 -16983.934,E2 -16983.934} C_VEL
LIN {X 0,Y 289.994,Z 349.387,A -85,B 0,C 180,E1 -16984.346,E2 -16984.346} C_VEL
LIN {X 0,Y 294.471,Z 382.673,A -85,B 0,C 180,E1 -16985.544,E2 -16985.544} C_VEL
LIN {X 0,Y 292.983,Z 448.296,A -85,B 0,C 180,E1 -16987.161,E2 -16987.161} C_VEL
LIN {X 0,Y 292.099,Z 462.037,A -85,B 0,C 180,E1 -16987.779,E2 -16987.779} C_VEL
LIN {X 0,Y 290.94,Z 475.039,A -85,B 0,C 180,E1 -16988.664,E2 -16988.664} C_VEL
LIN {X 0,Y 289.636,Z 486.87,A -85,B 0,C 180,E1 -16989.772,E2 -16989.772} C_VEL
LIN {X 0,Y 288.171,Z 498.268,A -85,B 0,C 180,E1 -16991.148,E2 -16991.148} C_VEL
LIN {X 0,Y 286.883,Z 508.539,A -85,B 0,C 180,E1 -16992.722,E2 -16992.722} C_VEL
LIN {X 0,Y 285.815,Z 516.944,A -85,B 0,C 180,E1 -16994.308,E2 -16994.308} C_VEL
LIN {X 0,Y 284.487,Z 526.049,A -85,B 0,C 180,E1 -16996.428,E2 -16996.428} C_VEL
LIN {X 0,Y 283.52,Z 533.378,A -85,B 0,C 180,E1 -16998.563,E2 -16998.563} C_VEL
LIN {X 0,Y 282.934,Z 539.236,A -85,B 0,C 180,E1 -17000.71,E2 -17000.71} C_VEL
LIN {X 0,Y 282.57,Z 543.83,A -85,B 0,C 180,E1 -17002.857,E2 -17002.857} C_VEL
LIN {X 0,Y 282.371,Z 546.718,A -85,B 0,C 180,E1 -17004.605,E2 -17004.605} C_VEL
LIN {X 0,Y 282.371,Z 549.774,A -85,B 0,C 180,E1 -17007.148,E2 -17007.148} C_VEL
LIN {X 0,Y 282.343,Z 550.879,A -85,B 0,C 180,E1 -17008.575,E2 -17008.575} C_VEL
LIN {X 0,Y 282.357,Z 551.569,A -85,B 0,C 180,E1 -17010.001,E2 -17010.001} C_VEL
LIN {X 0,Y 282.336,Z 551.869,A -85,B 0,C 180,E1 -17011.427,E2 -17011.427} C_VEL
LIN {X 0,Y 282.336,Z 551.785,A -85,B 0,C 180,E1 -17012.855,E2 -17012.855} C_VEL
LIN {X 0,Y 282.363,Z 550.645,A -85,B 0,C 180,E1 -17015.377,E2 -17015.377} C_VEL
LIN {X 0,Y 282.583,Z 549.077,A -85,B 0,C 180,E1 -17017.144,E2 -17017.144} C_VEL
LIN {X 0,Y 283.094,Z 546.345,A -85,B 0,C 180,E1 -17019.287,E2 -17019.287} C_VEL
LIN {X 0,Y 283.869,Z 542.612,A -85,B 0,C 180,E1 -17021.425,E2 -17021.425} C_VEL
LIN {X 0,Y 284.973,Z 537.785,A -85,B 0,C 180,E1 -17023.551,E2 -17023.551} C_VEL
LIN {X 0,Y 286.59,Z 531.717,A -85,B 0,C 180,E1 -17025.65,E2 -17025.65} C_VEL
LIN {X 0,Y 288.321,Z 524.477,A -85,B 0,C 180,E1 -17027.665,E2 -17027.665} C_VEL
LIN {X 0,Y 290.101,Z 516.703,A -85,B 0,C 180,E1 -17029.422,E2 -17029.422} C_VEL
LIN {X 0,Y 292.252,Z 507.238,A -85,B 0,C 180,E1 -17031.145,E2 -17031.145} C_VEL
LIN {X 0,Y 294.44,Z 496.921,A -85,B 0,C 180,E1 -17032.638,E2 -17032.638} C_VEL
LIN {X 0,Y 296.549,Z 485.492,A -85,B 0,C 180,E1 -17033.945,E2 -17033.945} C_VEL
LIN {X 0,Y 298.407,Z 473.525,A -85,B 0,C 180,E1 -17034.991,E2 -17034.991} C_VEL
LIN {X 0,Y 300.035,Z 460.237,A -85,B 0,C 180,E1 -17035.82,E2 -17035.82} C_VEL
LIN {X 0,Y 301.099,Z 447.024,A -85,B 0,C 180,E1 -17036.371,E2 -17036.371} C_VEL
LIN {X 0,Y 303.077,Z 385.383,A -85,B 0,C 180,E1 -17037.863,E2 -17037.863} C_VEL
LIN {X 0,Y 299.115,Z 363.201,A -85,B 0,C 180,E1 -17038.956,E2 -17038.956} C_VEL
LIN {X 0,Y 297.828,Z 358.069,A -85,B 0,C 180,E1 -17039.262,E2 -17039.262} C_VEL
LIN {X 0,Y 292.837,Z 346.79,A -85,B 0,C 180,E1 -17040.232,E2 -17040.232} C_VEL
LIN {X 0,Y 288.936,Z 338.557,A -85,B 0,C 180,E1 -17041.033,E2 -17041.033} C_VEL
LIN {X 0,Y 286.595,Z 328.636,A -85,B 0,C 180,E1 -17044.711,E2 -17044.711} C_VEL
LIN {X 0,Y 284.323,Z 320.069,A -85,B 0,C 180,E1 -17048.168,E2 -17048.168} C_VEL
LIN {X 0,Y 284.271,Z 320.074,A -85,B 0,C 180,E1 -17052.125,E2 -17052.125} C_VEL
LIN {X 0,Y 284.257,Z 320.074,A -85,B 0,C 180,E1 -17056.19,E2 -17056.19} C_VEL
LIN {X 0,Y 284.308,Z 320.07,A -85,B 0,C 180,E1 -17060.025,E2 -17060.025} C_VEL
LIN {X 0,Y 284.328,Z 320.066,A -85,B 0,C 180,E1 -17063.614,E2 -17063.614} C_VEL
LIN {X 0,Y 284.308,Z 320.065,A -85,B 0,C 180,E1 -17067.191,E2 -17067.191} C_VEL
LIN {X 0,Y 284.344,Z 320.066,A -85,B 0,C 180,E1 -17070.375,E2 -17070.375} C_VEL
LIN {X 0,Y 284.328,Z 320.067,A -85,B 0,C 180,E1 -17073.582,E2 -17073.582} C_VEL
LIN {X 0,Y 284.332,Z 320.065,A -85,B 0,C 180,E1 -17076.704,E2 -17076.704} C_VEL
LIN {X 0,Y 284.378,Z 320.057,A -85,B 0,C 180,E1 -17079.905,E2 -17079.905} C_VEL
LIN {X 0,Y 284.449,Z 320.048,A -85,B 0,C 180,E1 -17084.493,E2 -17084.493} C_VEL
LIN {X 0,Y 284.489,Z 320.041,A -85,B 0,C 180,E1 -17088.602,E2 -17088.602} C_VEL
LIN {X 0,Y 284.623,Z 320.019,A -85,B 0,C 180,E1 -17091.48,E2 -17091.48} C_VEL
LIN {X 0,Y 284.59,Z 320.029,A -85,B 0,C 180,E1 -17094.331,E2 -17094.331} C_VEL
LIN {X 0,Y 284.85,Z 319.997,A -85,B 0,C 180,E1 -17098.586,E2 -17098.586} C_VEL
LIN {X 0,Y 284.852,Z 319.992,A -85,B 0,C 180,E1 -17101.414,E2 -17101.414} C_VEL
LIN {X 0,Y 284.655,Z 320.024,A -85,B 0,C 180,E1 -17107.091,E2 -17107.091} C_VEL
LIN {X 0,Y 284.517,Z 320.036,A -85,B 0,C 180,E1 -17109.957,E2 -17109.957} C_VEL
LIN {X 0,Y 284.466,Z 320.043,A -85,B 0,C 180,E1 -17114.304,E2 -17114.304} C_VEL
LIN {X 0,Y 284.379,Z 320.057,A -85,B 0,C 180,E1 -17118.741,E2 -17118.741} C_VEL
LIN {X 0,Y 284.318,Z 320.06,A -85,B 0,C 180,E1 -17121.764,E2 -17121.764} C_VEL
LIN {X 0,Y 284.319,Z 320.061,A -85,B 0,C 180,E1 -17124.849,E2 -17124.849} C_VEL
LIN {X 0,Y 284.294,Z 320.065,A -85,B 0,C 180,E1 -17128.015,E2 -17128.015} C_VEL
LIN {X 0,Y 284.29,Z 320.067,A -85,B 0,C 180,E1 -17131.276,E2 -17131.276} C_VEL
LIN {X 0,Y 284.345,Z 320.063,A -85,B 0,C 180,E1 -17135.348,E2 -17135.348} C_VEL
LIN {X 0,Y 284.315,Z 320.07,A -85,B 0,C 180,E1 -17138.169,E2 -17138.169} C_VEL
LIN {X 0,Y 284.273,Z 320.072,A -85,B 0,C 180,E1 -17142.124,E2 -17142.124} C_VEL
LIN {X 0,Y 284.253,Z 320.194,A -85,B 0,C 180,E1 -17145.37,E2 -17145.37} C_VEL
LIN {X 0,Y 285.776,Z 325.714,A -85,B 0,C 180,E1 -17147.585,E2 -17147.585} C_VEL
LIN {X 0,Y 287.912,Z 329.594,A -85,B 0,C 180,E1 -17148.009,E2 -17148.009} C_VEL
LIN {X 0,Y 296.07,Z 345.37,A -85,B 0,C 180,E1 -17149.578,E2 -17149.578} C_VEL
LIN {X 0,Y 303.553,Z 362.114,A -85,B 0,C 180,E1 -17150.981,E2 -17150.981} C_VEL
LIN {X 0,Y 303.824,Z 362.876,A -85,B 0,C 180,E1 -17151.034,E2 -17151.034} C_VEL
LIN {X 0,Y 301.373,Z 433.32,A -85,B 0,C 180,E1 -17152.728,E2 -17152.728} C_VEL
LIN {X 0,Y 300.419,Z 445.892,A -85,B 0,C 180,E1 -17153.272,E2 -17153.272} C_VEL
LIN {X 0,Y 298.973,Z 458.947,A -85,B 0,C 180,E1 -17154.111,E2 -17154.111} C_VEL
LIN {X 0,Y 297.539,Z 469.62,A -85,B 0,C 180,E1 -17155.054,E2 -17155.054} C_VEL
LIN {X 0,Y 295.855,Z 480.154,A -85,B 0,C 180,E1 -17156.246,E2 -17156.246} C_VEL
LIN {X 0,Y 293.604,Z 491.245,A -85,B 0,C 180,E1 -17157.818,E2 -17157.818} C_VEL
LIN {X 0,Y 291.411,Z 501.041,A -85,B 0,C 180,E1 -17159.571,E2 -17159.571} C_VEL
LIN {X 0,Y 289.157,Z 510.38,A -85,B 0,C 180,E1 -17161.708,E2 -17161.708} C_VEL
LIN {X 0,Y 287.237,Z 517.847,A -85,B 0,C 180,E1 -17163.869,E2 -17163.869} C_VEL
LIN {X 0,Y 285.698,Z 523.768,A -85,B 0,C 180,E1 -17166.052,E2 -17166.052} C_VEL
LIN {X 0,Y 284.431,Z 528.371,A -85,B 0,C 180,E1 -17168.244,E2 -17168.244} C_VEL
LIN {X 0,Y 283.598,Z 531.69,A -85,B 0,C 180,E1 -17170.34,E2 -17170.34} C_VEL
LIN {X 0,Y 282.85,Z 534.247,A -85,B 0,C 180,E1 -17172.652,E2 -17172.652} C_VEL
LIN {X 0,Y 282.565,Z 535.287,A -85,B 0,C 180,E1 -17174.121,E2 -17174.121} C_VEL
LIN {X 0,Y 282.396,Z 536.068,A -85,B 0,C 180,E1 -17176.073,E2 -17176.073} C_VEL
LIN {X 0,Y 282.184,Z 535.987,A -85,B 0,C 180,E1 -17178.506,E2 -17178.506} C_VEL
LIN {X 0,Y 282.155,Z 535.384,A -85,B 0,C 180,E1 -17179.958,E2 -17179.958} C_VEL
LIN {X 0,Y 282.217,Z 534.388,A -85,B 0,C 180,E1 -17181.406,E2 -17181.406} C_VEL
LIN {X 0,Y 282.319,Z 532.997,A -85,B 0,C 180,E1 -17182.849,E2 -17182.849} C_VEL
LIN {X 0,Y 282.584,Z 530.595,A -85,B 0,C 180,E1 -17184.652,E2 -17184.652} C_VEL
LIN {X 0,Y 282.971,Z 526.112,A -85,B 0,C 180,E1 -17187.152,E2 -17187.152} C_VEL
LIN {X 0,Y 283.684,Z 520.024,A -85,B 0,C 180,E1 -17189.644,E2 -17189.644} C_VEL
LIN {X 0,Y 284.567,Z 513.374,A -85,B 0,C 180,E1 -17191.768,E2 -17191.768} C_VEL
LIN {X 0,Y 285.745,Z 505.125,A -85,B 0,C 180,E1 -17193.877,E2 -17193.877} C_VEL
LIN {X 0,Y 286.863,Z 496.678,A -85,B 0,C 180,E1 -17195.623,E2 -17195.623} C_VEL
LIN {X 0,Y 288.422,Z 486.2,A -85,B 0,C 180,E1 -17197.349,E2 -17197.349} C_VEL
LIN {X 0,Y 289.747,Z 475.843,A -85,B 0,C 180,E1 -17198.718,E2 -17198.718} C_VEL
LIN {X 0,Y 290.867,Z 464.533,A -85,B 0,C 180,E1 -17199.912,E2 -17199.912} C_VEL
LIN {X 0,Y 291.768,Z 452.932,A -85,B 0,C 180,E1 -17200.846,E2 -17200.846} C_VEL
LIN {X 0,Y 292.603,Z 439.559,A -85,B 0,C 180,E1 -17201.604,E2 -17201.604} C_VEL
LIN {X 0,Y 293.216,Z 426.28,A -85,B 0,C 180,E1 -17202.061,E2 -17202.061} C_VEL
LIN {X 0,Y 294.921,Z 357.961,A -85,B 0,C 180,E1 -17203.692,E2 -17203.692} C_VEL
LIN {X 0,Y 292.85,Z 345.684,A -85,B 0,C 180,E1 -17204.165,E2 -17204.165} C_VEL
LIN {X 0,Y 286.652,Z 328.084,A -85,B 0,C 180,E1 -17205.119,E2 -17205.119} C_VEL
LIN {X 0,Y 285.443,Z 324.836,A -85,B 0,C 180,E1 -17205.349,E2 -17205.349} C_VEL
LIN {X 0,Y 284.382,Z 320.063,A -85,B 0,C 180,E1 -17207.046,E2 -17207.046} C_VEL
LIN {X 0,Y 284.324,Z 320.07,A -85,B 0,C 180,E1 -17210.245,E2 -17210.245} C_VEL
LIN {X 0,Y 284.31,Z 320.07,A -85,B 0,C 180,E1 -17213.847,E2 -17213.847} C_VEL
LIN {X 0,Y 284.259,Z 320.076,A -85,B 0,C 180,E1 -17218.017,E2 -17218.017} C_VEL
LIN {X 0,Y 284.276,Z 320.071,A -85,B 0,C 180,E1 -17221.275,E2 -17221.275} C_VEL
LIN {X 0,Y 284.334,Z 320.064,A -85,B 0,C 180,E1 -17225.345,E2 -17225.345} C_VEL
LIN {X 0,Y 284.298,Z 320.07,A -85,B 0,C 180,E1 -17228.169,E2 -17228.169} C_VEL
LIN {X 0,Y 284.233,Z 320.075,A -85,B 0,C 180,E1 -17232.115,E2 -17232.115} C_VEL
LIN {X 0,Y 284.233,Z 320.074,A -85,B 0,C 180,E1 -17236.184,E2 -17236.184} C_VEL
LIN {X 0,Y 284.279,Z 320.07,A -85,B 0,C 180,E1 -17240.028,E2 -17240.028} C_VEL
LIN {X 0,Y 284.315,Z 320.062,A -85,B 0,C 180,E1 -17243.611,E2 -17243.611} C_VEL
LIN {X 0,Y 284.3,Z 320.068,A -85,B 0,C 180,E1 -17247.189,E2 -17247.189} C_VEL
LIN {X 0,Y 284.246,Z 320.069,A -85,B 0,C 180,E1 -17251.262,E2 -17251.262} C_VEL
LIN {X 0,Y 283.561,Z 320.157,A -85,B 0,C 180,E1 -17252.445,E2 -17252.445} C_VEL
LIN {X 0,Y 280.692,Z 320.509,A -85,B 0,C 180,E1 -17254.371,E2 -17254.371} C_VEL
LIN {X 0,Y 278.292,Z 320.816,A -85,B 0,C 180,E1 -17255.935,E2 -17255.935} C_VEL
LIN {X 0,Y 277.298,Z 320.94,A -85,B 0,C 180,E1 -17257.148,E2 -17257.148} C_VEL
LIN {X 0,Y 277.236,Z 320.95,A -85,B 0,C 180,E1 -17257.558,E2 -17257.558} C_VEL
LIN {X 0,Y 277.269,Z 320.944,A -85,B 0,C 180,E1 -17260.76,E2 -17260.76} C_VEL
LIN {X 0,Y 277.357,Z 320.924,A -85,B 0,C 180,E1 -17265.321,E2 -17265.321} C_VEL
LIN {X 0,Y 277.442,Z 320.926,A -85,B 0,C 180,E1 -17269.786,E2 -17269.786} C_VEL
LIN {X 0,Y 277.584,Z 320.901,A -85,B 0,C 180,E1 -17272.727,E2 -17272.727} C_VEL
LIN {X 0,Y 277.797,Z 320.881,A -85,B 0,C 180,E1 -17278.55,E2 -17278.55} C_VEL
LIN {X 0,Y 277.803,Z 320.877,A -85,B 0,C 180,E1 -17281.449,E2 -17281.449} C_VEL
LIN {X 0,Y 277.603,Z 320.899,A -85,B 0,C 180,E1 -17287.272,E2 -17287.272} C_VEL
LIN {X 0,Y 277.447,Z 320.923,A -85,B 0,C 180,E1 -17290.213,E2 -17290.213} C_VEL
LIN {X 0,Y 277.402,Z 320.924,A -85,B 0,C 180,E1 -17294.676,E2 -17294.676} C_VEL
LIN {X 0,Y 277.31,Z 320.942,A -85,B 0,C 180,E1 -17299.236,E2 -17299.236} C_VEL
LIN {X 0,Y 277.283,Z 320.941,A -85,B 0,C 180,E1 -17303.924,E2 -17303.924} C_VEL
LIN {X 0,Y 277.303,Z 320.94,A -85,B 0,C 180,E1 -17307.499,E2 -17307.499} C_VEL
LIN {X 0,Y 277.266,Z 320.944,A -85,B 0,C 180,E1 -17310.482,E2 -17310.482} C_VEL
LIN {X 0,Y 277.24,Z 320.949,A -85,B 0,C 180,E1 -17313.897,E2 -17313.897} C_VEL
LIN {X 0,Y 277.25,Z 320.949,A -85,B 0,C 180,E1 -17317.472,E2 -17317.472} C_VEL
LIN {X 0,Y 277.195,Z 320.954,A -85,B 0,C 180,E1 -17321.239,E2 -17321.239} C_VEL
LIN {X 0,Y 277.196,Z 320.955,A -85,B 0,C 180,E1 -17325.227,E2 -17325.227} C_VEL
LIN {X 0,Y 277.218,Z 320.953,A -85,B 0,C 180,E1 -17329.513,E2 -17329.513} C_VEL
LIN {X 0,Y 277.268,Z 320.947,A -85,B 0,C 180,E1 -17332.533,E2 -17332.533} C_VEL
LIN {X 0,Y 277.244,Z 320.954,A -85,B 0,C 180,E1 -17336.106,E2 -17336.106} C_VEL
LIN {X 0,Y 277.293,Z 321.087,A -85,B 0,C 180,E1 -17337.302,E2 -17337.302} C_VEL
LIN {X 0,Y 279.429,Z 330.885,A -85,B 0,C 180,E1 -17340.632,E2 -17340.632} C_VEL
LIN {X 0,Y 280.958,Z 339.176,A -85,B 0,C 180,E1 -17343.326,E2 -17343.326} C_VEL
LIN {X 0,Y 282.685,Z 345.681,A -85,B 0,C 180,E1 -17343.663,E2 -17343.663} C_VEL
LIN {X 0,Y 287.511,Z 381.006,A -85,B 0,C 180,E1 -17344.987,E2 -17344.987} C_VEL
LIN {X 0,Y 287.73,Z 386.979,A -85,B 0,C 180,E1 -17345.161,E2 -17345.161} C_VEL
LIN {X 0,Y 286.288,Z 448.134,A -85,B 0,C 180,E1 -17346.705,E2 -17346.705} C_VEL
LIN {X 0,Y 285.386,Z 461.644,A -85,B 0,C 180,E1 -17347.323,E2 -17347.323} C_VEL
LIN {X 0,Y 284.296,Z 473.644,A -85,B 0,C 180,E1 -17348.14,E2 -17348.14} C_VEL
LIN {X 0,Y 282.934,Z 485.771,A -85,B 0,C 180,E1 -17349.271,E2 -17349.271} C_VEL
LIN {X 0,Y 281.391,Z 497.331,A -85,B 0,C 180,E1 -17350.676,E2 -17350.676} C_VEL
LIN {X 0,Y 280.021,Z 507.76,A -85,B 0,C 180,E1 -17352.284,E2 -17352.284} C_VEL
LIN {X 0,Y 278.668,Z 517.928,A -85,B 0,C 180,E1 -17354.271,E2 -17354.271} C_VEL
LIN {X 0,Y 277.373,Z 526.841,A -85,B 0,C 180,E1 -17356.447,E2 -17356.447} C_VEL
LIN {X 0,Y 276.419,Z 533.96,A -85,B 0,C 180,E1 -17358.637,E2 -17358.637} C_VEL
LIN {X 0,Y 275.722,Z 540.451,A -85,B 0,C 180,E1 -17361.204,E2 -17361.204} C_VEL
LIN {X 0,Y 275.405,Z 544.716,A -85,B 0,C 180,E1 -17363.407,E2 -17363.407} C_VEL
LIN {X 0,Y 275.252,Z 547.896,A -85,B 0,C 180,E1 -17365.608,E2 -17365.608} C_VEL
LIN {X 0,Y 275.279,Z 549.476,A -85,B 0,C 180,E1 -17367.074,E2 -17367.074} C_VEL
LIN {X 0,Y 275.268,Z 550.626,A -85,B 0,C 180,E1 -17368.538,E2 -17368.538} C_VEL
LIN {X 0,Y 275.279,Z 551.337,A -85,B 0,C 180,E1 -17370.001,E2 -17370.001} C_VEL
LIN {X 0,Y 275.26,Z 551.66,A -85,B 0,C 180,E1 -17371.464,E2 -17371.464} C_VEL
LIN {X 0,Y 275.245,Z 551.597,A -85,B 0,C 180,E1 -17372.928,E2 -17372.928} C_VEL
LIN {X 0,Y 275.254,Z 550.657,A -85,B 0,C 180,E1 -17375.265,E2 -17375.265} C_VEL
LIN {X 0,Y 275.517,Z 548.979,A -85,B 0,C 180,E1 -17377.329,E2 -17377.329} C_VEL
LIN {X 0,Y 276.056,Z 546.295,A -85,B 0,C 180,E1 -17379.526,E2 -17379.526} C_VEL
LIN {X 0,Y 276.902,Z 542.613,A -85,B 0,C 180,E1 -17381.716,E2 -17381.716} C_VEL
LIN {X 0,Y 278.054,Z 537.84,A -85,B 0,C 180,E1 -17383.894,E2 -17383.894} C_VEL
LIN {X 0,Y 280.096,Z 530.716,A -85,B 0,C 180,E1 -17386.397,E2 -17386.397} C_VEL
LIN {X 0,Y 281.927,Z 523.088,A -85,B 0,C 180,E1 -17388.506,E2 -17388.506} C_VEL
LIN {X 0,Y 284.261,Z 513.331,A -85,B 0,C 180,E1 -17390.63,E2 -17390.63} C_VEL
LIN {X 0,Y 286.643,Z 503.375,A -85,B 0,C 180,E1 -17392.337,E2 -17392.337} C_VEL
LIN {X 0,Y 289.047,Z 492.13,A -85,B 0,C 180,E1 -17393.843,E2 -17393.843} C_VEL
LIN {X 0,Y 290.961,Z 481.15,A -85,B 0,C 180,E1 -17395.006,E2 -17395.006} C_VEL
LIN {X 0,Y 292.85,Z 468.977,A -85,B 0,C 180,E1 -17395.976,E2 -17395.976} C_VEL
LIN {X 0,Y 294.234,Z 456.229,A -85,B 0,C 180,E1 -17396.703,E2 -17396.703} C_VEL
LIN {X 0,Y 295.232,Z 442.48,A -85,B 0,C 180,E1 -17397.189,E2 -17397.189} C_VEL
LIN {X 0,Y 296.968,Z 386.105,A -85,B 0,C 180,E1 -17398.574,E2 -17398.574} C_VEL
LIN {X 0,Y 293.041,Z 363.962,A -85,B 0,C 180,E1 -17399.706,E2 -17399.706} C_VEL
LIN {X 0,Y 291.991,Z 360.426,A -85,B 0,C 180,E1 -17399.946,E2 -17399.946} C_VEL
LIN {X 0,Y 287.41,Z 350.216,A -85,B 0,C 180,E1 -17400.868,E2 -17400.868} C_VEL
LIN {X 0,Y 281.667,Z 338.269,A -85,B 0,C 180,E1 -17402.095,E2 -17402.095} C_VEL
LIN {X 0,Y 279.322,Z 328.349,A -85,B 0,C 180,E1 -17405.937,E2 -17405.937} C_VEL
LIN {X 0,Y 277.252,Z 320.948,A -85,B 0,C 180,E1 -17409.094,E2 -17409.094} C_VEL
LIN {X 0,Y 277.211,Z 320.953,A -85,B 0,C 180,E1 -17413.199,E2 -17413.199} C_VEL
LIN {X 0,Y 277.217,Z 320.954,A -85,B 0,C 180,E1 -17417.326,E2 -17417.326} C_VEL
LIN {X 0,Y 277.259,Z 320.941,A -85,B 0,C 180,E1 -17421.795,E2 -17421.795} C_VEL
LIN {X 0,Y 277.281,Z 320.94,A -85,B 0,C 180,E1 -17424.341,E2 -17424.341} C_VEL
LIN {X 0,Y 277.242,Z 320.942,A -85,B 0,C 180,E1 -17427.836,E2 -17427.836} C_VEL
LIN {X 0,Y 277.247,Z 320.943,A -85,B 0,C 180,E1 -17431.208,E2 -17431.208} C_VEL
LIN {X 0,Y 277.279,Z 320.943,A -85,B 0,C 180,E1 -17434.476,E2 -17434.476} C_VEL
LIN {X 0,Y 277.266,Z 320.946,A -85,B 0,C 180,E1 -17437.653,E2 -17437.653} C_VEL
LIN {X 0,Y 277.307,Z 320.94,A -85,B 0,C 180,E1 -17440.764,E2 -17440.764} C_VEL
LIN {X 0,Y 277.412,Z 320.928,A -85,B 0,C 180,E1 -17445.325,E2 -17445.325} C_VEL
LIN {X 0,Y 277.462,Z 320.92,A -85,B 0,C 180,E1 -17449.787,E2 -17449.787} C_VEL
LIN {X 0,Y 277.629,Z 320.894,A -85,B 0,C 180,E1 -17452.729,E2 -17452.729} C_VEL
LIN {X 0,Y 277.816,Z 320.873,A -85,B 0,C 180,E1 -17458.551,E2 -17458.551} C_VEL
LIN {X 0,Y 277.818,Z 320.869,A -85,B 0,C 180,E1 -17461.45,E2 -17461.45} C_VEL
LIN {X 0,Y 277.613,Z 320.901,A -85,B 0,C 180,E1 -17467.272,E2 -17467.272} C_VEL
LIN {X 0,Y 277.46,Z 320.916,A -85,B 0,C 180,E1 -17470.213,E2 -17470.213} C_VEL
LIN {X 0,Y 277.413,Z 320.925,A -85,B 0,C 180,E1 -17474.676,E2 -17474.676} C_VEL
LIN {X 0,Y 277.328,Z 320.94,A -85,B 0,C 180,E1 -17479.235,E2 -17479.235} C_VEL
LIN {X 0,Y 277.29,Z 320.94,A -85,B 0,C 180,E1 -17483.924,E2 -17483.924} C_VEL
LIN {X 0,Y 277.284,Z 320.94,A -85,B 0,C 180,E1 -17487.487,E2 -17487.487} C_VEL
LIN {X 0,Y 277.251,Z 320.947,A -85,B 0,C 180,E1 -17490.473,E2 -17490.473} C_VEL
LIN {X 0,Y 277.25,Z 320.946,A -85,B 0,C 180,E1 -17493.896,E2 -17493.896} C_VEL
LIN {X 0,Y 277.271,Z 320.943,A -85,B 0,C 180,E1 -17497.469,E2 -17497.469} C_VEL
LIN {X 0,Y 277.213,Z 320.955,A -85,B 0,C 180,E1 -17501.237,E2 -17501.237} C_VEL
LIN {X 0,Y 277.211,Z 320.964,A -85,B 0,C 180,E1 -17504.428,E2 -17504.428} C_VEL
LIN {X 0,Y 278.626,Z 326.05,A -85,B 0,C 180,E1 -17506.523,E2 -17506.523} C_VEL
LIN {X 0,Y 287.8,Z 343.054,A -85,B 0,C 180,E1 -17508.399,E2 -17508.399} C_VEL
LIN {X 0,Y 295.122,Z 358.458,A -85,B 0,C 180,E1 -17509.831,E2 -17509.831} C_VEL
LIN {X 0,Y 297.762,Z 364.66,A -85,B 0,C 180,E1 -17510.344,E2 -17510.344} C_VEL
LIN {X 0,Y 295.284,Z 433.675,A -85,B 0,C 180,E1 -17512.04,E2 -17512.04} C_VEL
LIN {X 0,Y 294.259,Z 446.174,A -85,B 0,C 180,E1 -17512.587,E2 -17512.587} C_VEL
LIN {X 0,Y 292.774,Z 459.206,A -85,B 0,C 180,E1 -17513.442,E2 -17513.442} C_VEL
LIN {X 0,Y 291.285,Z 469.86,A -85,B 0,C 180,E1 -17514.402,E2 -17514.402} C_VEL
LIN {X 0,Y 289.471,Z 480.566,A -85,B 0,C 180,E1 -17515.638,E2 -17515.638} C_VEL
LIN {X 0,Y 287.185,Z 491.464,A -85,B 0,C 180,E1 -17517.217,E2 -17517.217} C_VEL
LIN {X 0,Y 285.083,Z 500.343,A -85,B 0,C 180,E1 -17518.821,E2 -17518.821} C_VEL
LIN {X 0,Y 283.068,Z 508.474,A -85,B 0,C 180,E1 -17520.635,E2 -17520.635} C_VEL
LIN {X 0,Y 280.982,Z 516.341,A -85,B 0,C 180,E1 -17522.839,E2 -17522.839} C_VEL
LIN {X 0,Y 279.319,Z 522.273,A -85,B 0,C 180,E1 -17524.933,E2 -17524.933} C_VEL
LIN {X 0,Y 277.635,Z 528.242,A -85,B 0,C 180,E1 -17527.684,E2 -17527.684} C_VEL
LIN {X 0,Y 276.625,Z 531.945,A -85,B 0,C 180,E1 -17530.058,E2 -17530.058} C_VEL
LIN {X 0,Y 275.881,Z 534.284,A -85,B 0,C 180,E1 -17532.199,E2 -17532.199} C_VEL
LIN {X 0,Y 275.546,Z 535.389,A -85,B 0,C 180,E1 -17533.705,E2 -17533.705} C_VEL
LIN {X 0,Y 275.324,Z 536.274,A -85,B 0,C 180,E1 -17535.933,E2 -17535.933} C_VEL
LIN {X 0,Y 275.113,Z 536.24,A -85,B 0,C 180,E1 -17538.207,E2 -17538.207} C_VEL
LIN {X 0,Y 275.05,Z 535.684,A -85,B 0,C 180,E1 -17539.696,E2 -17539.696} C_VEL
LIN {X 0,Y 275.105,Z 534.729,A -85,B 0,C 180,E1 -17541.182,E2 -17541.182} C_VEL
LIN {X 0,Y 275.216,Z 533.378,A -85,B 0,C 180,E1 -17542.663,E2 -17542.663} C_VEL
LIN {X 0,Y 275.494,Z 530.755,A -85,B 0,C 180,E1 -17544.721,E2 -17544.721} C_VEL
LIN {X 0,Y 275.866,Z 526.66,A -85,B 0,C 180,E1 -17547.078,E2 -17547.078} C_VEL
LIN {X 0,Y 276.473,Z 521.662,A -85,B 0,C 180,E1 -17549.271,E2 -17549.271} C_VEL
LIN {X 0,Y 277.272,Z 515.394,A -85,B 0,C 180,E1 -17551.451,E2 -17551.451} C_VEL
LIN {X 0,Y 278.512,Z 507.525,A -85,B 0,C 180,E1 -17553.616,E2 -17553.616} C_VEL
LIN {X 0,Y 279.818,Z 497.762,A -85,B 0,C 180,E1 -17555.765,E2 -17555.765} C_VEL
LIN {X 0,Y 281.265,Z 488.685,A -85,B 0,C 180,E1 -17557.356,E2 -17557.356} C_VEL
LIN {X 0,Y 282.789,Z 477.425,A -85,B 0,C 180,E1 -17558.935,E2 -17558.935} C_VEL
LIN {X 0,Y 283.943,Z 466.442,A -85,B 0,C 180,E1 -17560.156,E2 -17560.156} C_VEL
LIN {X 0,Y 284.95,Z 454.296,A -85,B 0,C 180,E1 -17561.199,E2 -17561.199} C_VEL
LIN {X 0,Y 285.804,Z 441.493,A -85,B 0,C 180,E1 -17561.974,E2 -17561.974} C_VEL
LIN {X 0,Y 286.482,Z 427.864,A -85,B 0,C 180,E1 -17562.484,E2 -17562.484} C_VEL
LIN {X 0,Y 288.283,Z 358.854,A -85,B 0,C 180,E1 -17564.172,E2 -17564.172} C_VEL
LIN {X 0,Y 286.312,Z 347.308,A -85,B 0,C 180,E1 -17564.634,E2 -17564.634} C_VEL
LIN {X 0,Y 280.103,Z 330.083,A -85,B 0,C 180,E1 -17565.612,E2 -17565.612} C_VEL
LIN {X 0,Y 278.242,Z 325.122,A -85,B 0,C 180,E1 -17565.927,E2 -17565.927} C_VEL
LIN {X 0,Y 277.314,Z 320.945,A -85,B 0,C 180,E1 -17567.418,E2 -17567.418} C_VEL
LIN {X 0,Y 277.263,Z 320.949,A -85,B 0,C 180,E1 -17570.784,E2 -17570.784} C_VEL
LIN {X 0,Y 277.252,Z 320.951,A -85,B 0,C 180,E1 -17574.137,E2 -17574.137} C_VEL
LIN {X 0,Y 277.235,Z 320.949,A -85,B 0,C 180,E1 -17577.467,E2 -17577.467} C_VEL
LIN {X 0,Y 277.227,Z 320.952,A -85,B 0,C 180,E1 -17580.464,E2 -17580.464} C_VEL
LIN {X 0,Y 277.244,Z 320.947,A -85,B 0,C 180,E1 -17583.894,E2 -17583.894} C_VEL
LIN {X 0,Y 277.257,Z 320.946,A -85,B 0,C 180,E1 -17587.469,E2 -17587.469} C_VEL
LIN {X 0,Y 277.18,Z 320.955,A -85,B 0,C 180,E1 -17591.24,E2 -17591.24} C_VEL
LIN {X 0,Y 277.169,Z 320.956,A -85,B 0,C 180,E1 -17595.231,E2 -17595.231} C_VEL
LIN {X 0,Y 277.179,Z 320.954,A -85,B 0,C 180,E1 -17598.757,E2 -17598.757} C_VEL
LIN {X 0,Y 277.249,Z 320.946,A -85,B 0,C 180,E1 -17602.527,E2 -17602.527} C_VEL
LIN {X 0,Y 277.24,Z 320.943,A -85,B 0,C 180,E1 -17606.103,E2 -17606.103} C_VEL
LIN {X 0,Y 277.222,Z 320.953,A -85,B 0,C 180,E1 -17609.533,E2 -17609.533} C_VEL
LIN {X 0,Y 277.243,Z 320.943,A -85,B 0,C 180,E1 -17612.851,E2 -17612.851} C_VEL
LIN {X 0,Y 277.253,Z 320.945,A -85,B 0,C 180,E1 -17616.072,E2 -17616.072} C_VEL
LIN {X 0,Y 277.236,Z 320.95,A -85,B 0,C 180,E1 -17617.558,E2 -17617.558} C_VEL
LIN {X 0,Y 276.608,Z 321.037,A -85,B 0,C 180,E1 -17618.772,E2 -17618.772} C_VEL
LIN {X 0,Y 273.746,Z 321.394,A -85,B 0,C 180,E1 -17620.748,E2 -17620.748} C_VEL
LIN {X 0,Y 271.329,Z 321.686,A -85,B 0,C 180,E1 -17622.354,E2 -17622.354} C_VEL
LIN {X 0,Y 270.346,Z 321.801,A -85,B 0,C 180,E1 -17623.6,E2 -17623.6} C_VEL
LIN {X 0,Y 270.297,Z 321.803,A -85,B 0,C 180,E1 -17624.021,E2 -17624.021} C_VEL
LIN {X 0,Y 270.338,Z 321.809,A -85,B 0,C 180,E1 -17627.996,E2 -17627.996} C_VEL
LIN {X 0,Y 270.492,Z 321.788,A -85,B 0,C 180,E1 -17631.031,E2 -17631.031} C_VEL
LIN {X 0,Y 270.501,Z 321.782,A -85,B 0,C 180,E1 -17634.034,E2 -17634.034} C_VEL
LIN {X 0,Y 270.762,Z 321.757,A -85,B 0,C 180,E1 -17638.512,E2 -17638.512} C_VEL
LIN {X 0,Y 270.768,Z 321.754,A -85,B 0,C 180,E1 -17641.487,E2 -17641.487} C_VEL
LIN {X 0,Y 270.563,Z 321.775,A -85,B 0,C 180,E1 -17647.462,E2 -17647.462} C_VEL
LIN {X 0,Y 270.399,Z 321.803,A -85,B 0,C 180,E1 -17650.482,E2 -17650.482} C_VEL
LIN {X 0,Y 270.361,Z 321.797,A -85,B 0,C 180,E1 -17655.067,E2 -17655.067} C_VEL
LIN {X 0,Y 270.25,Z 321.819,A -85,B 0,C 180,E1 -17659.759,E2 -17659.759} C_VEL
LIN {X 0,Y 270.226,Z 321.821,A -85,B 0,C 180,E1 -17664.59,E2 -17664.59} C_VEL
LIN {X 0,Y 270.237,Z 321.818,A -85,B 0,C 180,E1 -17667.912,E2 -17667.912} C_VEL
LIN {X 0,Y 270.178,Z 321.831,A -85,B 0,C 180,E1 -17671.349,E2 -17671.349} C_VEL
LIN {X 0,Y 270.192,Z 321.827,A -85,B 0,C 180,E1 -17674.907,E2 -17674.907} C_VEL
LIN {X 0,Y 270.192,Z 321.826,A -85,B 0,C 180,E1 -17678.711,E2 -17678.711} C_VEL
LIN {X 0,Y 270.155,Z 321.828,A -85,B 0,C 180,E1 -17683.249,E2 -17683.249} C_VEL
LIN {X 0,Y 270.167,Z 321.832,A -85,B 0,C 180,E1 -17687.443,E2 -17687.443} C_VEL
LIN {X 0,Y 270.203,Z 321.827,A -85,B 0,C 180,E1 -17691.375,E2 -17691.375} C_VEL
LIN {X 0,Y 270.199,Z 321.828,A -85,B 0,C 180,E1 -17695.096,E2 -17695.096} C_VEL
LIN {X 0,Y 270.234,Z 321.892,A -85,B 0,C 180,E1 -17696.829,E2 -17696.829} C_VEL
LIN {X 0,Y 272.598,Z 332.909,A -85,B 0,C 180,E1 -17700.671,E2 -17700.671} C_VEL
LIN {X 0,Y 273.758,Z 339.154,A -85,B 0,C 180,E1 -17702.721,E2 -17702.721} C_VEL
LIN {X 0,Y 276.216,Z 347.146,A -85,B 0,C 180,E1 -17703.159,E2 -17703.159} C_VEL
LIN {X 0,Y 280.979,Z 382.591,A -85,B 0,C 180,E1 -17704.523,E2 -17704.523} C_VEL
LIN {X 0,Y 280.998,Z 392.695,A -85,B 0,C 180,E1 -17704.798,E2 -17704.798} C_VEL
LIN {X 0,Y 279.624,Z 447.577,A -85,B 0,C 180,E1 -17706.211,E2 -17706.211} C_VEL
LIN {X 0,Y 278.681,Z 461.248,A -85,B 0,C 180,E1 -17706.844,E2 -17706.844} C_VEL
LIN {X 0,Y 277.565,Z 473.301,A -85,B 0,C 180,E1 -17707.68,E2 -17707.68} C_VEL
LIN {X 0,Y 276.303,Z 484.68,A -85,B 0,C 180,E1 -17708.75,E2 -17708.75} C_VEL
LIN {X 0,Y 274.629,Z 496.394,A -85,B 0,C 180,E1 -17710.181,E2 -17710.181} C_VEL
LIN {X 0,Y 273.195,Z 506.953,A -85,B 0,C 180,E1 -17711.826,E2 -17711.826} C_VEL
LIN {X 0,Y 272.075,Z 515.581,A -85,B 0,C 180,E1 -17713.494,E2 -17713.494} C_VEL
LIN {X 0,Y 270.858,Z 523.505,A -85,B 0,C 180,E1 -17715.347,E2 -17715.347} C_VEL
LIN {X 0,Y 269.674,Z 531.221,A -85,B 0,C 180,E1 -17717.585,E2 -17717.585} C_VEL
LIN {X 0,Y 268.85,Z 538.336,A -85,B 0,C 180,E1 -17720.218,E2 -17720.218} C_VEL
LIN {X 0,Y 268.421,Z 543.045,A -85,B 0,C 180,E1 -17722.479,E2 -17722.479} C_VEL
LIN {X 0,Y 268.179,Z 546.671,A -85,B 0,C 180,E1 -17724.774,E2 -17724.774} C_VEL
LIN {X 0,Y 268.189,Z 549.175,A -85,B 0,C 180,E1 -17726.997,E2 -17726.997} C_VEL
LIN {X 0,Y 268.194,Z 550.364,A -85,B 0,C 180,E1 -17728.5,E2 -17728.5} C_VEL
LIN {X 0,Y 268.202,Z 551.105,A -85,B 0,C 180,E1 -17730.001,E2 -17730.001} C_VEL
LIN {X 0,Y 268.186,Z 551.45,A -85,B 0,C 180,E1 -17731.503,E2 -17731.503} C_VEL
LIN {X 0,Y 268.157,Z 551.409,A -85,B 0,C 180,E1 -17733.006,E2 -17733.006} C_VEL
LIN {X 0,Y 268.167,Z 550.627,A -85,B 0,C 180,E1 -17735.197,E2 -17735.197} C_VEL
LIN {X 0,Y 268.458,Z 548.882,A -85,B 0,C 180,E1 -17737.522,E2 -17737.522} C_VEL
LIN {X 0,Y 269.033,Z 546.245,A -85,B 0,C 180,E1 -17739.777,E2 -17739.777} C_VEL
LIN {X 0,Y 269.925,Z 542.613,A -85,B 0,C 180,E1 -17742.023,E2 -17742.023} C_VEL
LIN {X 0,Y 271.153,Z 537.894,A -85,B 0,C 180,E1 -17744.255,E2 -17744.255} C_VEL
LIN {X 0,Y 273.283,Z 530.829,A -85,B 0,C 180,E1 -17746.818,E2 -17746.818} C_VEL
LIN {X 0,Y 275.333,Z 522.75,A -85,B 0,C 180,E1 -17749.112,E2 -17749.112} C_VEL
LIN {X 0,Y 277.64,Z 513.641,A -85,B 0,C 180,E1 -17751.145,E2 -17751.145} C_VEL
LIN {X 0,Y 280.126,Z 503.795,A -85,B 0,C 180,E1 -17752.885,E2 -17752.885} C_VEL
LIN {X 0,Y 282.344,Z 494.132,A -85,B 0,C 180,E1 -17754.25,E2 -17754.25} C_VEL
LIN {X 0,Y 284.304,Z 483.723,A -85,B 0,C 180,E1 -17755.437,E2 -17755.437} C_VEL
LIN {X 0,Y 286.37,Z 471.209,A -85,B 0,C 180,E1 -17756.511,E2 -17756.511} C_VEL
LIN {X 0,Y 287.977,Z 458.034,A -85,B 0,C 180,E1 -17757.331,E2 -17757.331} C_VEL
LIN {X 0,Y 289.062,Z 444.932,A -85,B 0,C 180,E1 -17757.846,E2 -17757.846} C_VEL
LIN {X 0,Y 291.01,Z 387.358,A -85,B 0,C 180,E1 -17759.289,E2 -17759.289} C_VEL
LIN {X 0,Y 287.046,Z 364.897,A -85,B 0,C 180,E1 -17760.479,E2 -17760.479} C_VEL
LIN {X 0,Y 282.561,Z 354.611,A -85,B 0,C 180,E1 -17761.421,E2 -17761.421} C_VEL
LIN {X 0,Y 275.986,Z 341.441,A -85,B 0,C 180,E1 -17762.823,E2 -17762.823} C_VEL
LIN {X 0,Y 274.425,Z 338.066,A -85,B 0,C 180,E1 -17763.199,E2 -17763.199} C_VEL
LIN {X 0,Y 272.213,Z 329.095,A -85,B 0,C 180,E1 -17766.836,E2 -17766.836} C_VEL
LIN {X 0,Y 270.177,Z 321.83,A -85,B 0,C 180,E1 -17770.085,E2 -17770.085} C_VEL
LIN {X 0,Y 270.167,Z 321.83,A -85,B 0,C 180,E1 -17773.249,E2 -17773.249} C_VEL
LIN {X 0,Y 270.174,Z 321.832,A -85,B 0,C 180,E1 -17777.442,E2 -17777.442} C_VEL
LIN {X 0,Y 270.209,Z 321.82,A -85,B 0,C 180,E1 -17781.375,E2 -17781.375} C_VEL
LIN {X 0,Y 270.201,Z 321.822,A -85,B 0,C 180,E1 -17785.095,E2 -17785.095} C_VEL
LIN {X 0,Y 270.186,Z 321.827,A -85,B 0,C 180,E1 -17789.137,E2 -17789.137} C_VEL
LIN {X 0,Y 270.224,Z 321.819,A -85,B 0,C 180,E1 -17792.164,E2 -17792.164} C_VEL
LIN {X 0,Y 270.233,Z 321.817,A -85,B 0,C 180,E1 -17795.541,E2 -17795.541} C_VEL
LIN {X 0,Y 270.254,Z 321.817,A -85,B 0,C 180,E1 -17800.241,E2 -17800.241} C_VEL
LIN {X 0,Y 270.371,Z 321.802,A -85,B 0,C 180,E1 -17804.934,E2 -17804.934} C_VEL
LIN {X 0,Y 270.414,Z 321.798,A -85,B 0,C 180,E1 -17809.518,E2 -17809.518} C_VEL
LIN {X 0,Y 270.586,Z 321.769,A -85,B 0,C 180,E1 -17812.538,E2 -17812.538} C_VEL
LIN {X 0,Y 270.78,Z 321.75,A -85,B 0,C 180,E1 -17818.513,E2 -17818.513} C_VEL
LIN {X 0,Y 270.784,Z 321.745,A -85,B 0,C 180,E1 -17821.488,E2 -17821.488} C_VEL
LIN {X 0,Y 270.573,Z 321.778,A -85,B 0,C 180,E1 -17827.463,E2 -17827.463} C_VEL
LIN {X 0,Y 270.413,Z 321.797,A -85,B 0,C 180,E1 -17830.483,E2 -17830.483} C_VEL
LIN {X 0,Y 270.38,Z 321.806,A -85,B 0,C 180,E1 -17835.066,E2 -17835.066} C_VEL
LIN {X 0,Y 270.265,Z 321.818,A -85,B 0,C 180,E1 -17839.759,E2 -17839.759} C_VEL
LIN {X 0,Y 270.231,Z 321.816,A -85,B 0,C 180,E1 -17844.59,E2 -17844.59} C_VEL
LIN {X 0,Y 270.212,Z 321.819,A -85,B 0,C 180,E1 -17847.916,E2 -17847.916} C_VEL
LIN {X 0,Y 270.177,Z 321.824,A -85,B 0,C 180,E1 -17851.35,E2 -17851.35} C_VEL
LIN {X 0,Y 270.206,Z 321.821,A -85,B 0,C 180,E1 -17854.906,E2 -17854.906} C_VEL
LIN {X 0,Y 270.201,Z 321.829,A -85,B 0,C 180,E1 -17858.71,E2 -17858.71} C_VEL
LIN {X 0,Y 270.17,Z 321.833,A -85,B 0,C 180,E1 -17863.249,E2 -17863.249} C_VEL
LIN {X 0,Y 270.178,Z 321.916,A -85,B 0,C 180,E1 -17863.495,E2 -17863.495} C_VEL
LIN {X 0,Y 271.317,Z 326.136,A -85,B 0,C 180,E1 -17865.353,E2 -17865.353} C_VEL
LIN {X 0,Y 273.684,Z 330.246,A -85,B 0,C 180,E1 -17865.876,E2 -17865.876} C_VEL
LIN {X 0,Y 282.431,Z 346.387,A -85,B 0,C 180,E1 -17867.733,E2 -17867.733} C_VEL
LIN {X 0,Y 289.886,Z 362.248,A -85,B 0,C 180,E1 -17869.255,E2 -17869.255} C_VEL
LIN {X 0,Y 291.732,Z 366.646,A -85,B 0,C 180,E1 -17869.628,E2 -17869.628} C_VEL
LIN {X 0,Y 289.29,Z 433.311,A -85,B 0,C 180,E1 -17871.295,E2 -17871.295} C_VEL
LIN {X 0,Y 288.143,Z 446.61,A -85,B 0,C 180,E1 -17871.882,E2 -17871.882} C_VEL
LIN {X 0,Y 286.618,Z 459.494,A -85,B 0,C 180,E1 -17872.745,E2 -17872.745} C_VEL
LIN {X 0,Y 285.049,Z 470.122,A -85,B 0,C 180,E1 -17873.719,E2 -17873.719} C_VEL
LIN {X 0,Y 282.913,Z 482.114,A -85,B 0,C 180,E1 -17875.154,E2 -17875.154} C_VEL
LIN {X 0,Y 280.53,Z 492.801,A -85,B 0,C 180,E1 -17876.768,E2 -17876.768} C_VEL
LIN {X 0,Y 278.37,Z 501.48,A -85,B 0,C 180,E1 -17878.407,E2 -17878.407} C_VEL
LIN {X 0,Y 276.225,Z 509.629,A -85,B 0,C 180,E1 -17880.318,E2 -17880.318} C_VEL
LIN {X 0,Y 274.112,Z 517.124,A -85,B 0,C 180,E1 -17882.515,E2 -17882.515} C_VEL
LIN {X 0,Y 272.131,Z 523.88,A -85,B 0,C 180,E1 -17885.047,E2 -17885.047} C_VEL
LIN {X 0,Y 270.858,Z 528.086,A -85,B 0,C 180,E1 -17887.094,E2 -17887.094} C_VEL
LIN {X 0,Y 269.625,Z 532.224,A -85,B 0,C 180,E1 -17889.781,E2 -17889.781} C_VEL
LIN {X 0,Y 268.914,Z 534.304,A -85,B 0,C 180,E1 -17891.722,E2 -17891.722} C_VEL
LIN {X 0,Y 268.538,Z 535.489,A -85,B 0,C 180,E1 -17893.268,E2 -17893.268} C_VEL
LIN {X 0,Y 268.251,Z 536.479,A -85,B 0,C 180,E1 -17895.786,E2 -17895.786} C_VEL
LIN {X 0,Y 268.056,Z 536.466,A -85,B 0,C 180,E1 -17897.891,E2 -17897.891} C_VEL
LIN {X 0,Y 267.952,Z 535.985,A -85,B 0,C 180,E1 -17899.419,E2 -17899.419} C_VEL
LIN {X 0,Y 268.01,Z 535.068,A -85,B 0,C 180,E1 -17900.947,E2 -17900.947} C_VEL
LIN {X 0,Y 268.093,Z 533.758,A -85,B 0,C 180,E1 -17902.467,E2 -17902.467} C_VEL
LIN {X 0,Y 268.364,Z 531.521,A -85,B 0,C 180,E1 -17904.365,E2 -17904.365} C_VEL
LIN {X 0,Y 268.766,Z 527.207,A -85,B 0,C 180,E1 -17907.001,E2 -17907.001} C_VEL
LIN {X 0,Y 269.37,Z 522.303,A -85,B 0,C 180,E1 -17909.251,E2 -17909.251} C_VEL
LIN {X 0,Y 270.163,Z 516.142,A -85,B 0,C 180,E1 -17911.49,E2 -17911.49} C_VEL
LIN {X 0,Y 271.455,Z 508.447,A -85,B 0,C 180,E1 -17913.71,E2 -17913.71} C_VEL
LIN {X 0,Y 272.773,Z 498.829,A -85,B 0,C 180,E1 -17915.914,E2 -17915.914} C_VEL
LIN {X 0,Y 274.249,Z 489.927,A -85,B 0,C 180,E1 -17917.546,E2 -17917.546} C_VEL
LIN {X 0,Y 275.837,Z 479.005,A -85,B 0,C 180,E1 -17919.162,E2 -17919.162} C_VEL
LIN {X 0,Y 277.188,Z 466.599,A -85,B 0,C 180,E1 -17920.591,E2 -17920.591} C_VEL
LIN {X 0,Y 278.235,Z 454.443,A -85,B 0,C 180,E1 -17921.657,E2 -17921.657} C_VEL
LIN {X 0,Y 279.12,Z 441.611,A -85,B 0,C 180,E1 -17922.449,E2 -17922.449} C_VEL
LIN {X 0,Y 279.821,Z 427.931,A -85,B 0,C 180,E1 -17922.971,E2 -17922.971} C_VEL
LIN {X 0,Y 281.636,Z 359.515,A -85,B 0,C 180,E1 -17924.683,E2 -17924.683} C_VEL
LIN {X 0,Y 279.879,Z 349.348,A -85,B 0,C 180,E1 -17925.104,E2 -17925.104} C_VEL
LIN {X 0,Y 273.901,Z 332.741,A -85,B 0,C 180,E1 -17926.079,E2 -17926.079} C_VEL
LIN {X 0,Y 271.017,Z 325.329,A -85,B 0,C 180,E1 -17926.573,E2 -17926.573} C_VEL
LIN {X 0,Y 270.246,Z 321.826,A -85,B 0,C 180,E1 -17927.889,E2 -17927.889} C_VEL
LIN {X 0,Y 270.192,Z 321.829,A -85,B 0,C 180,E1 -17931.354,E2 -17931.354} C_VEL
LIN {X 0,Y 270.184,Z 321.83,A -85,B 0,C 180,E1 -17934.593,E2 -17934.593} C_VEL
LIN {X 0,Y 270.183,Z 321.829,A -85,B 0,C 180,E1 -17937.917,E2 -17937.917} C_VEL
LIN {X 0,Y 270.167,Z 321.829,A -85,B 0,C 180,E1 -17941.349,E2 -17941.349} C_VEL
LIN {X 0,Y 270.197,Z 321.827,A -85,B 0,C 180,E1 -17944.904,E2 -17944.904} C_VEL
LIN {X 0,Y 270.195,Z 321.829,A -85,B 0,C 180,E1 -17948.709,E2 -17948.709} C_VEL
LIN {X 0,Y 270.144,Z 321.834,A -85,B 0,C 180,E1 -17953.243,E2 -17953.243} C_VEL
LIN {X 0,Y 270.146,Z 321.828,A -85,B 0,C 180,E1 -17957.436,E2 -17957.436} C_VEL
LIN {X 0,Y 270.203,Z 321.826,A -85,B 0,C 180,E1 -17961.373,E2 -17961.373} C_VEL
LIN {X 0,Y 270.192,Z 321.82,A -85,B 0,C 180,E1 -17965.093,E2 -17965.093} C_VEL
LIN {X 0,Y 270.165,Z 321.831,A -85,B 0,C 180,E1 -17969.14,E2 -17969.14} C_VEL
LIN {X 0,Y 270.181,Z 321.822,A -85,B 0,C 180,E1 -17972.176,E2 -17972.176} C_VEL
LIN {X 0,Y 270.177,Z 321.823,A -85,B 0,C 180,E1 -17975.562,E2 -17975.562} C_VEL
LIN {X 0,Y 270.212,Z 321.824,A -85,B 0,C 180,E1 -17980.237,E2 -17980.237} C_VEL
LIN {X 0,Y 270.297,Z 321.803,A -85,B 0,C 180,E1 -17984.021,E2 -17984.021} C_VEL
LIN {X 0,Y 270.035,Z 321.834,A -85,B 0,C 180,E1 -17984.853,E2 -17984.853} C_VEL
LIN {X 0,Y 268.714,Z 322.006,A -85,B 0,C 180,E1 -17986.08,E2 -17986.08} C_VEL
LIN {X 0,Y 264.415,Z 322.545,A -85,B 0,C 180,E1 -17988.937,E2 -17988.937} C_VEL
LIN {X 0,Y 263.467,Z 322.666,A -85,B 0,C 180,E1 -17990.216,E2 -17990.216} C_VEL
LIN {X 0,Y 263.439,Z 322.666,A -85,B 0,C 180,E1 -17990.648,E2 -17990.648} C_VEL
LIN {X 0,Y 263.472,Z 322.658,A -85,B 0,C 180,E1 -17993.875,E2 -17993.875} C_VEL
LIN {X 0,Y 263.726,Z 322.633,A -85,B 0,C 180,E1 -17998.473,E2 -17998.473} C_VEL
LIN {X 0,Y 263.731,Z 322.63,A -85,B 0,C 180,E1 -18001.527,E2 -18001.527} C_VEL
LIN {X 0,Y 263.525,Z 322.651,A -85,B 0,C 180,E1 -18007.663,E2 -18007.663} C_VEL
LIN {X 0,Y 263.338,Z 322.684,A -85,B 0,C 180,E1 -18010.767,E2 -18010.767} C_VEL
LIN {X 0,Y 263.303,Z 322.674,A -85,B 0,C 180,E1 -18015.481,E2 -18015.481} C_VEL
LIN {X 0,Y 263.23,Z 322.694,A -85,B 0,C 180,E1 -18020.309,E2 -18020.309} C_VEL
LIN {X 0,Y 263.179,Z 322.703,A -85,B 0,C 180,E1 -18025.294,E2 -18025.294} C_VEL
LIN {X 0,Y 263.148,Z 322.701,A -85,B 0,C 180,E1 -18028.733,E2 -18028.733} C_VEL
LIN {X 0,Y 263.126,Z 322.704,A -85,B 0,C 180,E1 -18032.289,E2 -18032.289} C_VEL
LIN {X 0,Y 263.17,Z 322.7,A -85,B 0,C 180,E1 -18036.762,E2 -18036.762} C_VEL
LIN {X 0,Y 263.097,Z 322.711,A -85,B 0,C 180,E1 -18039.874,E2 -18039.874} C_VEL
LIN {X 0,Y 263.097,Z 322.713,A -85,B 0,C 180,E1 -18043.989,E2 -18043.989} C_VEL
LIN {X 0,Y 263.119,Z 322.71,A -85,B 0,C 180,E1 -18048.108,E2 -18048.108} C_VEL
LIN {X 0,Y 263.159,Z 322.706,A -85,B 0,C 180,E1 -18052.105,E2 -18052.105} C_VEL
LIN {X 0,Y 263.205,Z 322.768,A -85,B 0,C 180,E1 -18056.356,E2 -18056.356} C_VEL
LIN {X 0,Y 265.254,Z 332.24,A -85,B 0,C 180,E1 -18059.776,E2 -18059.776} C_VEL
LIN {X 0,Y 266.538,Z 338.974,A -85,B 0,C 180,E1 -18062.058,E2 -18062.058} C_VEL
LIN {X 0,Y 269.795,Z 348.971,A -85,B 0,C 180,E1 -18062.645,E2 -18062.645} C_VEL
LIN {X 0,Y 274.483,Z 384.291,A -85,B 0,C 180,E1 -18064.044,E2 -18064.044} C_VEL
LIN {X 0,Y 272.931,Z 447.724,A -85,B 0,C 180,E1 -18065.721,E2 -18065.721} C_VEL
LIN {X 0,Y 271.956,Z 461.606,A -85,B 0,C 180,E1 -18066.388,E2 -18066.388} C_VEL
LIN {X 0,Y 270.734,Z 474.047,A -85,B 0,C 180,E1 -18067.287,E2 -18067.287} C_VEL
LIN {X 0,Y 269.2,Z 486.765,A -85,B 0,C 180,E1 -18068.563,E2 -18068.563} C_VEL
LIN {X 0,Y 267.553,Z 498.071,A -85,B 0,C 180,E1 -18070.034,E2 -18070.034} C_VEL
LIN {X 0,Y 266.25,Z 507.226,A -85,B 0,C 180,E1 -18071.535,E2 -18071.535} C_VEL
LIN {X 0,Y 264.967,Z 516.608,A -85,B 0,C 180,E1 -18073.434,E2 -18073.434} C_VEL
LIN {X 0,Y 263.727,Z 524.304,A -85,B 0,C 180,E1 -18075.337,E2 -18075.337} C_VEL
LIN {X 0,Y 262.513,Z 531.832,A -85,B 0,C 180,E1 -18077.634,E2 -18077.634} C_VEL
LIN {X 0,Y 261.804,Z 537.879,A -85,B 0,C 180,E1 -18079.952,E2 -18079.952} C_VEL
LIN {X 0,Y 261.352,Z 542.644,A -85,B 0,C 180,E1 -18082.274,E2 -18082.274} C_VEL
LIN {X 0,Y 261.084,Z 546.645,A -85,B 0,C 180,E1 -18084.866,E2 -18084.866} C_VEL
LIN {X 0,Y 261.101,Z 548.874,A -85,B 0,C 180,E1 -18086.915,E2 -18086.915} C_VEL
LIN {X 0,Y 261.122,Z 550.092,A -85,B 0,C 180,E1 -18088.459,E2 -18088.459} C_VEL
LIN {X 0,Y 261.128,Z 550.874,A -85,B 0,C 180,E1 -18090.001,E2 -18090.001} C_VEL
LIN {X 0,Y 261.113,Z 551.24,A -85,B 0,C 180,E1 -18091.543,E2 -18091.543} C_VEL
LIN {X 0,Y 261.067,Z 550.819,A -85,B 0,C 180,E1 -18094.633,E2 -18094.633} C_VEL
LIN {X 0,Y 261.166,Z 550.014,A -85,B 0,C 180,E1 -18096.18,E2 -18096.18} C_VEL
LIN {X 0,Y 261.787,Z 547.158,A -85,B 0,C 180,E1 -18099.27,E2 -18099.27} C_VEL
LIN {X 0,Y 262.592,Z 543.912,A -85,B 0,C 180,E1 -18101.581,E2 -18101.581} C_VEL
LIN {X 0,Y 263.729,Z 539.622,A -85,B 0,C 180,E1 -18103.878,E2 -18103.878} C_VEL
LIN {X 0,Y 265.791,Z 533.162,A -85,B 0,C 180,E1 -18106.515,E2 -18106.515} C_VEL
LIN {X 0,Y 267.829,Z 525.918,A -85,B 0,C 180,E1 -18108.807,E2 -18108.807} C_VEL
LIN {X 0,Y 270.156,Z 517.337,A -85,B 0,C 180,E1 -18110.96,E2 -18110.96} C_VEL
LIN {X 0,Y 272.861,Z 507.389,A -85,B 0,C 180,E1 -18112.929,E2 -18112.929} C_VEL
LIN {X 0,Y 275.246,Z 497.259,A -85,B 0,C 180,E1 -18114.515,E2 -18114.515} C_VEL
LIN {X 0,Y 277.631,Z 486.042,A -85,B 0,C 180,E1 -18115.892,E2 -18115.892} C_VEL
LIN {X 0,Y 279.549,Z 475.42,A -85,B 0,C 180,E1 -18116.907,E2 -18116.907} C_VEL
LIN {X 0,Y 281.445,Z 462.593,A -85,B 0,C 180,E1 -18117.818,E2 -18117.818} C_VEL
LIN {X 0,Y 282.712,Z 449.815,A -85,B 0,C 180,E1 -18118.433,E2 -18118.433} C_VEL
LIN {X 0,Y 283.577,Z 431.515,A -85,B 0,C 180,E1 -18118.955,E2 -18118.955} C_VEL
LIN {X 0,Y 285.045,Z 388.047,A -85,B 0,C 180,E1 -18120.058,E2 -18120.058} C_VEL
LIN {X 0,Y 281.419,Z 367.623,A -85,B 0,C 180,E1 -18121.186,E2 -18121.186} C_VEL
LIN {X 0,Y 277.23,Z 358.021,A -85,B 0,C 180,E1 -18122.104,E2 -18122.104} C_VEL
LIN {X 0,Y 269.416,Z 342.245,A -85,B 0,C 180,E1 -18123.854,E2 -18123.854} C_VEL
LIN {X 0,Y 267.137,Z 337.74,A -85,B 0,C 180,E1 -18124.433,E2 -18124.433} C_VEL
LIN {X 0,Y 265.049,Z 329.503,A -85,B 0,C 180,E1 -18127.94,E2 -18127.94} C_VEL
LIN {X 0,Y 263.142,Z 322.705,A -85,B 0,C 180,E1 -18131.163,E2 -18131.163} C_VEL
LIN {X 0,Y 263.106,Z 322.708,A -85,B 0,C 180,E1 -18133.989,E2 -18133.989} C_VEL
LIN {X 0,Y 263.126,Z 322.705,A -85,B 0,C 180,E1 -18138.407,E2 -18138.407} C_VEL
LIN {X 0,Y 263.16,Z 322.698,A -85,B 0,C 180,E1 -18142.103,E2 -18142.103} C_VEL
LIN {X 0,Y 263.153,Z 322.704,A -85,B 0,C 180,E1 -18145.886,E2 -18145.886} C_VEL
LIN {X 0,Y 263.129,Z 322.709,A -85,B 0,C 180,E1 -18149.504,E2 -18149.504} C_VEL
LIN {X 0,Y 263.149,Z 322.706,A -85,B 0,C 180,E1 -18152.998,E2 -18152.998} C_VEL
LIN {X 0,Y 263.151,Z 322.703,A -85,B 0,C 180,E1 -18156.384,E2 -18156.384} C_VEL
LIN {X 0,Y 263.238,Z 322.688,A -85,B 0,C 180,E1 -18159.691,E2 -18159.691} C_VEL
LIN {X 0,Y 263.313,Z 322.681,A -85,B 0,C 180,E1 -18164.52,E2 -18164.52} C_VEL
LIN {X 0,Y 263.354,Z 322.675,A -85,B 0,C 180,E1 -18169.234,E2 -18169.234} C_VEL
LIN {X 0,Y 263.546,Z 322.645,A -85,B 0,C 180,E1 -18172.338,E2 -18172.338} C_VEL
LIN {X 0,Y 263.744,Z 322.627,A -85,B 0,C 180,E1 -18178.473,E2 -18178.473} C_VEL
LIN {X 0,Y 263.749,Z 322.621,A -85,B 0,C 180,E1 -18181.527,E2 -18181.527} C_VEL
LIN {X 0,Y 263.535,Z 322.655,A -85,B 0,C 180,E1 -18187.663,E2 -18187.663} C_VEL
LIN {X 0,Y 263.355,Z 322.679,A -85,B 0,C 180,E1 -18190.767,E2 -18190.767} C_VEL
LIN {X 0,Y 263.327,Z 322.684,A -85,B 0,C 180,E1 -18195.48,E2 -18195.48} C_VEL
LIN {X 0,Y 263.242,Z 322.691,A -85,B 0,C 180,E1 -18200.309,E2 -18200.309} C_VEL
LIN {X 0,Y 263.176,Z 322.693,A -85,B 0,C 180,E1 -18205.295,E2 -18205.295} C_VEL
LIN {X 0,Y 263.142,Z 322.698,A -85,B 0,C 180,E1 -18208.735,E2 -18208.735} C_VEL
LIN {X 0,Y 263.132,Z 322.702,A -85,B 0,C 180,E1 -18212.289,E2 -18212.289} C_VEL
LIN {X 0,Y 263.195,Z 322.698,A -85,B 0,C 180,E1 -18216.766,E2 -18216.766} C_VEL
LIN {X 0,Y 263.128,Z 322.707,A -85,B 0,C 180,E1 -18221.593,E2 -18221.593} C_VEL
LIN {X 0,Y 263.185,Z 322.927,A -85,B 0,C 180,E1 -18222.528,E2 -18222.528} C_VEL
LIN {X 0,Y 264.174,Z 326.559,A -85,B 0,C 180,E1 -18224.133,E2 -18224.133} C_VEL
LIN {X 0,Y 271.525,Z 339.295,A -85,B 0,C 180,E1 -18225.822,E2 -18225.822} C_VEL
LIN {X 0,Y 278.907,Z 353.3,A -85,B 0,C 180,E1 -18227.426,E2 -18227.426} C_VEL
LIN {X 0,Y 285.718,Z 368.649,A -85,B 0,C 180,E1 -18228.879,E2 -18228.879} C_VEL
LIN {X 0,Y 283.364,Z 432.484,A -85,B 0,C 180,E1 -18230.502,E2 -18230.502} C_VEL
LIN {X 0,Y 282.249,Z 445.462,A -85,B 0,C 180,E1 -18231.058,E2 -18231.058} C_VEL
LIN {X 0,Y 280.685,Z 458.636,A -85,B 0,C 180,E1 -18231.932,E2 -18231.932} C_VEL
LIN {X 0,Y 279.145,Z 468.591,A -85,B 0,C 180,E1 -18232.825,E2 -18232.825} C_VEL
LIN {X 0,Y 277.213,Z 479.682,A -85,B 0,C 180,E1 -18234.106,E2 -18234.106} C_VEL
LIN {X 0,Y 274.705,Z 490.847,A -85,B 0,C 180,E1 -18235.746,E2 -18235.746} C_VEL
LIN {X 0,Y 272.16,Z 500.808,A -85,B 0,C 180,E1 -18237.599,E2 -18237.599} C_VEL
LIN {X 0,Y 269.724,Z 509.564,A -85,B 0,C 180,E1 -18239.654,E2 -18239.654} C_VEL
LIN {X 0,Y 267.615,Z 516.774,A -85,B 0,C 180,E1 -18241.789,E2 -18241.789} C_VEL
LIN {X 0,Y 265.656,Z 522.963,A -85,B 0,C 180,E1 -18244.091,E2 -18244.091} C_VEL
LIN {X 0,Y 264.078,Z 527.934,A -85,B 0,C 180,E1 -18246.471,E2 -18246.471} C_VEL
LIN {X 0,Y 263.223,Z 530.57,A -85,B 0,C 180,E1 -18248.049,E2 -18248.049} C_VEL
LIN {X 0,Y 262.572,Z 532.672,A -85,B 0,C 180,E1 -18249.637,E2 -18249.637} C_VEL
LIN {X 0,Y 261.986,Z 534.326,A -85,B 0,C 180,E1 -18251.221,E2 -18251.221} C_VEL
LIN {X 0,Y 261.544,Z 535.562,A -85,B 0,C 180,E1 -18252.807,E2 -18252.807} C_VEL
LIN {X 0,Y 261.156,Z 536.685,A -85,B 0,C 180,E1 -18255.652,E2 -18255.652} C_VEL
LIN {X 0,Y 260.974,Z 536.687,A -85,B 0,C 180,E1 -18257.558,E2 -18257.558} C_VEL
LIN {X 0,Y 260.86,Z 536.269,A -85,B 0,C 180,E1 -18259.128,E2 -18259.128} C_VEL
LIN {X 0,Y 260.89,Z 535.408,A -85,B 0,C 180,E1 -18260.697,E2 -18260.697} C_VEL
LIN {X 0,Y 260.997,Z 534.137,A -85,B 0,C 180,E1 -18262.261,E2 -18262.261} C_VEL
LIN {X 0,Y 261.282,Z 531.708,A -85,B 0,C 180,E1 -18264.409,E2 -18264.409} C_VEL
LIN {X 0,Y 261.671,Z 527.754,A -85,B 0,C 180,E1 -18266.92,E2 -18266.92} C_VEL
LIN {X 0,Y 262.27,Z 522.944,A -85,B 0,C 180,E1 -18269.231,E2 -18269.231} C_VEL
LIN {X 0,Y 263.06,Z 516.886,A -85,B 0,C 180,E1 -18271.53,E2 -18271.53} C_VEL
LIN {X 0,Y 264.37,Z 509.334,A -85,B 0,C 180,E1 -18273.81,E2 -18273.81} C_VEL
LIN {X 0,Y 265.501,Z 501.644,A -85,B 0,C 180,E1 -18275.696,E2 -18275.696} C_VEL
LIN {X 0,Y 266.932,Z 492.253,A -85,B 0,C 180,E1 -18277.563,E2 -18277.563} C_VEL
LIN {X 0,Y 268.67,Z 481.779,A -85,B 0,C 180,E1 -18279.219,E2 -18279.219} C_VEL
LIN {X 0,Y 270.087,Z 470.201,A -85,B 0,C 180,E1 -18280.683,E2 -18280.683} C_VEL
LIN {X 0,Y 271.254,Z 457.925,A -85,B 0,C 180,E1 -18281.867,E2 -18281.867} C_VEL
LIN {X 0,Y 272.244,Z 444.999,A -85,B 0,C 180,E1 -18282.769,E2 -18282.769} C_VEL
LIN {X 0,Y 272.969,Z 432.371,A -85,B 0,C 180,E1 -18283.35,E2 -18283.35} C_VEL
LIN {X 0,Y 275.082,Z 360.61,A -85,B 0,C 180,E1 -18285.197,E2 -18285.197} C_VEL
LIN {X 0,Y 273.464,Z 351.327,A -85,B 0,C 180,E1 -18285.595,E2 -18285.595} C_VEL
LIN {X 0,Y 267.265,Z 334.118,A -85,B 0,C 180,E1 -18286.647,E2 -18286.647} C_VEL
LIN {X 0,Y 263.851,Z 325.504,A -85,B 0,C 180,E1 -18287.26,E2 -18287.26} C_VEL
LIN {X 0,Y 263.199,Z 322.704,A -85,B 0,C 180,E1 -18288.384,E2 -18288.384} C_VEL
LIN {X 0,Y 263.129,Z 322.71,A -85,B 0,C 180,E1 -18291.957,E2 -18291.957} C_VEL
LIN {X 0,Y 263.124,Z 322.708,A -85,B 0,C 180,E1 -18295.298,E2 -18295.298} C_VEL
LIN {X 0,Y 263.117,Z 322.709,A -85,B 0,C 180,E1 -18298.735,E2 -18298.735} C_VEL
LIN {X 0,Y 263.125,Z 322.71,A -85,B 0,C 180,E1 -18302.288,E2 -18302.288} C_VEL
LIN {X 0,Y 263.176,Z 322.703,A -85,B 0,C 180,E1 -18306.76,E2 -18306.76} C_VEL
LIN {X 0,Y 263.088,Z 322.709,A -85,B 0,C 180,E1 -18309.874,E2 -18309.874} C_VEL
LIN {X 0,Y 263.073,Z 322.713,A -85,B 0,C 180,E1 -18313.993,E2 -18313.993} C_VEL
LIN {X 0,Y 263.075,Z 322.708,A -85,B 0,C 180,E1 -18318.416,E2 -18318.416} C_VEL
LIN {X 0,Y 263.152,Z 322.701,A -85,B 0,C 180,E1 -18322.101,E2 -18322.101} C_VEL
LIN {X 0,Y 263.146,Z 322.698,A -85,B 0,C 180,E1 -18325.884,E2 -18325.884} C_VEL
LIN {X 0,Y 263.103,Z 322.712,A -85,B 0,C 180,E1 -18329.5,E2 -18329.5} C_VEL
LIN {X 0,Y 263.107,Z 322.704,A -85,B 0,C 180,E1 -18332.993,E2 -18332.993} C_VEL
LIN {X 0,Y 263.111,Z 322.705,A -85,B 0,C 180,E1 -18336.38,E2 -18336.38} C_VEL
LIN {X 0,Y 263.2,Z 322.701,A -85,B 0,C 180,E1 -18339.688,E2 -18339.688} C_VEL
LIN {X 0,Y 263.281,Z 322.674,A -85,B 0,C 180,E1 -18344.517,E2 -18344.517} C_VEL
LIN {X 0,Y 263.318,Z 322.682,A -85,B 0,C 180,E1 -18349.232,E2 -18349.232} C_VEL
LIN {X 0,Y 263.439,Z 322.666,A -85,B 0,C 180,E1 -18350.648,E2 -18350.648} C_VEL
LIN {X 0,Y 262.877,Z 322.741,A -85,B 0,C 180,E1 -18351.923,E2 -18351.923} C_VEL
LIN {X 0,Y 259.988,Z 323.099,A -85,B 0,C 180,E1 -18353.999,E2 -18353.999} C_VEL
LIN {X 0,Y 257.52,Z 323.4,A -85,B 0,C 180,E1 -18355.689,E2 -18355.689} C_VEL
LIN {X 0,Y 256.545,Z 323.52,A -85,B 0,C 180,E1 -18357.002,E2 -18357.002} C_VEL
LIN {X 0,Y 256.515,Z 323.524,A -85,B 0,C 180,E1 -18357.446,E2 -18357.446} C_VEL
LIN {X 0,Y 256.688,Z 323.509,A -85,B 0,C 180,E1 -18360,E2 -18360} C_VEL
LIN {X 0,Y 256.693,Z 323.507,A -85,B 0,C 180,E1 -18361.569,E2 -18361.569} C_VEL
LIN {X 0,Y 256.453,Z 323.526,A -85,B 0,C 180,E1 -18366.293,E2 -18366.293} C_VEL
LIN {X 0,Y 256.395,Z 323.544,A -85,B 0,C 180,E1 -18369.466,E2 -18369.466} C_VEL
LIN {X 0,Y 256.225,Z 323.563,A -85,B 0,C 180,E1 -18374.292,E2 -18374.292} C_VEL
LIN {X 0,Y 256.166,Z 323.571,A -85,B 0,C 180,E1 -18377.565,E2 -18377.565} C_VEL
LIN {X 0,Y 256.135,Z 323.58,A -85,B 0,C 180,E1 -18381.111,E2 -18381.111} C_VEL
LIN {X 0,Y 256.16,Z 323.577,A -85,B 0,C 180,E1 -18385.128,E2 -18385.128} C_VEL
LIN {X 0,Y 256.092,Z 323.584,A -85,B 0,C 180,E1 -18389.602,E2 -18389.602} C_VEL
LIN {X 0,Y 256.061,Z 323.586,A -85,B 0,C 180,E1 -18393.294,E2 -18393.294} C_VEL
LIN {X 0,Y 256.104,Z 323.582,A -85,B 0,C 180,E1 -18397.27,E2 -18397.27} C_VEL
LIN {X 0,Y 256.045,Z 323.587,A -85,B 0,C 180,E1 -18401.205,E2 -18401.205} C_VEL
LIN {X 0,Y 256.049,Z 323.592,A -85,B 0,C 180,E1 -18405.532,E2 -18405.532} C_VEL
LIN {X 0,Y 256.05,Z 323.589,A -85,B 0,C 180,E1 -18408.798,E2 -18408.798} C_VEL
LIN {X 0,Y 256.134,Z 323.579,A -85,B 0,C 180,E1 -18412.87,E2 -18412.87} C_VEL
LIN {X 0,Y 256.125,Z 323.608,A -85,B 0,C 180,E1 -18415.839,E2 -18415.839} C_VEL
LIN {X 0,Y 258.416,Z 334.051,A -85,B 0,C 180,E1 -18419.724,E2 -18419.724} C_VEL
LIN {X 0,Y 259.313,Z 338.811,A -85,B 0,C 180,E1 -18421.356,E2 -18421.356} C_VEL
LIN {X 0,Y 263.423,Z 350.843,A -85,B 0,C 180,E1 -18422.111,E2 -18422.111} C_VEL
LIN {X 0,Y 267.921,Z 385.386,A -85,B 0,C 180,E1 -18423.518,E2 -18423.518} C_VEL
LIN {X 0,Y 266.301,Z 447.13,A -85,B 0,C 180,E1 -18425.18,E2 -18425.18} C_VEL
LIN {X 0,Y 265.384,Z 460.384,A -85,B 0,C 180,E1 -18425.819,E2 -18425.819} C_VEL
LIN {X 0,Y 264.196,Z 472.561,A -85,B 0,C 180,E1 -18426.692,E2 -18426.692} C_VEL
LIN {X 0,Y 262.85,Z 484.04,A -85,B 0,C 180,E1 -18427.812,E2 -18427.812} C_VEL
LIN {X 0,Y 261.069,Z 495.808,A -85,B 0,C 180,E1 -18429.311,E2 -18429.311} C_VEL
LIN {X 0,Y 259.636,Z 505.314,A -85,B 0,C 180,E1 -18430.841,E2 -18430.841} C_VEL
LIN {X 0,Y 258.355,Z 514.149,A -85,B 0,C 180,E1 -18432.59,E2 -18432.59} C_VEL
LIN {X 0,Y 257.006,Z 522.25,A -85,B 0,C 180,E1 -18434.538,E2 -18434.538} C_VEL
LIN {X 0,Y 255.722,Z 530.179,A -85,B 0,C 180,E1 -18436.896,E2 -18436.896} C_VEL
LIN {X 0,Y 255.018,Z 535.557,A -85,B 0,C 180,E1 -18438.879,E2 -18438.879} C_VEL
LIN {X 0,Y 254.445,Z 540.792,A -85,B 0,C 180,E1 -18441.263,E2 -18441.263} C_VEL
LIN {X 0,Y 254.081,Z 544.837,A -85,B 0,C 180,E1 -18443.649,E2 -18443.649} C_VEL
LIN {X 0,Y 253.973,Z 546.918,A -85,B 0,C 180,E1 -18445.239,E2 -18445.239} C_VEL
LIN {X 0,Y 253.997,Z 548.571,A -85,B 0,C 180,E1 -18446.829,E2 -18446.829} C_VEL
LIN {X 0,Y 254.05,Z 549.814,A -85,B 0,C 180,E1 -18448.416,E2 -18448.416} C_VEL
LIN {X 0,Y 254.056,Z 550.64,A -85,B 0,C 180,E1 -18450.001,E2 -18450.001} C_VEL
LIN {X 0,Y 254.018,Z 551.03,A -85,B 0,C 180,E1 -18451.587,E2 -18451.587} C_VEL
LIN {X 0,Y 253.974,Z 550.654,A -85,B 0,C 180,E1 -18454.763,E2 -18454.763} C_VEL
LIN {X 0,Y 254.081,Z 549.889,A -85,B 0,C 180,E1 -18456.353,E2 -18456.353} C_VEL
LIN {X 0,Y 254.77,Z 547.089,A -85,B 0,C 180,E1 -18459.528,E2 -18459.528} C_VEL
LIN {X 0,Y 255.615,Z 543.893,A -85,B 0,C 180,E1 -18461.901,E2 -18461.901} C_VEL
LIN {X 0,Y 256.827,Z 539.658,A -85,B 0,C 180,E1 -18464.259,E2 -18464.259} C_VEL
LIN {X 0,Y 258.991,Z 533.257,A -85,B 0,C 180,E1 -18466.962,E2 -18466.962} C_VEL
LIN {X 0,Y 261.059,Z 526.318,A -85,B 0,C 180,E1 -18469.251,E2 -18469.251} C_VEL
LIN {X 0,Y 263.544,Z 517.612,A -85,B 0,C 180,E1 -18471.512,E2 -18471.512} C_VEL
LIN {X 0,Y 266.038,Z 508.735,A -85,B 0,C 180,E1 -18473.346,E2 -18473.346} C_VEL
LIN {X 0,Y 268.829,Z 497.808,A -85,B 0,C 180,E1 -18475.14,E2 -18475.14} C_VEL
LIN {X 0,Y 271.288,Z 486.762,A -85,B 0,C 180,E1 -18476.545,E2 -18476.545} C_VEL
LIN {X 0,Y 273.637,Z 474.4,A -85,B 0,C 180,E1 -18477.744,E2 -18477.744} C_VEL
LIN {X 0,Y 275.417,Z 462.637,A -85,B 0,C 180,E1 -18478.586,E2 -18478.586} C_VEL
LIN {X 0,Y 276.721,Z 450.357,A -85,B 0,C 180,E1 -18479.195,E2 -18479.195} C_VEL
LIN {X 0,Y 277.59,Z 433.15,A -85,B 0,C 180,E1 -18479.71,E2 -18479.71} C_VEL
LIN {X 0,Y 279.151,Z 389.023,A -85,B 0,C 180,E1 -18480.851,E2 -18480.851} C_VEL
LIN {X 0,Y 275.831,Z 370.353,A -85,B 0,C 180,E1 -18481.925,E2 -18481.925} C_VEL
LIN {X 0,Y 272.091,Z 361.673,A -85,B 0,C 180,E1 -18482.782,E2 -18482.782} C_VEL
LIN {X 0,Y 264.52,Z 346.325,A -85,B 0,C 180,E1 -18484.55,E2 -18484.55} C_VEL
LIN {X 0,Y 259.89,Z 337.518,A -85,B 0,C 180,E1 -18485.716,E2 -18485.716} C_VEL
LIN {X 0,Y 257.846,Z 329.741,A -85,B 0,C 180,E1 -18489.206,E2 -18489.206} C_VEL
LIN {X 0,Y 256.055,Z 323.589,A -85,B 0,C 180,E1 -18492.277,E2 -18492.277} C_VEL
LIN {X 0,Y 256.051,Z 323.588,A -85,B 0,C 180,E1 -18496.671,E2 -18496.671} C_VEL
LIN {X 0,Y 256.073,Z 323.583,A -85,B 0,C 180,E1 -18500.858,E2 -18500.858} C_VEL
LIN {X 0,Y 256.13,Z 323.58,A -85,B 0,C 180,E1 -18502.867,E2 -18502.867} C_VEL
LIN {X 0,Y 256.068,Z 323.587,A -85,B 0,C 180,E1 -18506.707,E2 -18506.707} C_VEL
LIN {X 0,Y 256.058,Z 323.588,A -85,B 0,C 180,E1 -18510.393,E2 -18510.393} C_VEL
LIN {X 0,Y 256.163,Z 323.57,A -85,B 0,C 180,E1 -18514.875,E2 -18514.875} C_VEL
LIN {X 0,Y 256.15,Z 323.569,A -85,B 0,C 180,E1 -18519.104,E2 -18519.104} C_VEL
LIN {X 0,Y 256.233,Z 323.56,A -85,B 0,C 180,E1 -18524.081,E2 -18524.081} C_VEL
LIN {X 0,Y 256.295,Z 323.553,A -85,B 0,C 180,E1 -18528.934,E2 -18528.934} C_VEL
LIN {X 0,Y 256.506,Z 323.52,A -85,B 0,C 180,E1 -18532.126,E2 -18532.126} C_VEL
LIN {X 0,Y 256.463,Z 323.527,A -85,B 0,C 180,E1 -18536.858,E2 -18536.858} C_VEL
LIN {X 0,Y 256.746,Z 323.49,A -85,B 0,C 180,E1 -18540,E2 -18540} C_VEL
LIN {X 0,Y 256.487,Z 323.531,A -85,B 0,C 180,E1 -18543.142,E2 -18543.142} C_VEL
LIN {X 0,Y 256.498,Z 323.531,A -85,B 0,C 180,E1 -18547.875,E2 -18547.875} C_VEL
LIN {X 0,Y 256.298,Z 323.56,A -85,B 0,C 180,E1 -18551.067,E2 -18551.067} C_VEL
LIN {X 0,Y 256.24,Z 323.559,A -85,B 0,C 180,E1 -18554.291,E2 -18554.291} C_VEL
LIN {X 0,Y 256.181,Z 323.563,A -85,B 0,C 180,E1 -18557.564,E2 -18557.564} C_VEL
LIN {X 0,Y 256.145,Z 323.569,A -85,B 0,C 180,E1 -18561.111,E2 -18561.111} C_VEL
LIN {X 0,Y 256.163,Z 323.566,A -85,B 0,C 180,E1 -18565.125,E2 -18565.125} C_VEL
LIN {X 0,Y 256.061,Z 323.585,A -85,B 0,C 180,E1 -18569.607,E2 -18569.607} C_VEL
LIN {X 0,Y 256.07,Z 323.589,A -85,B 0,C 180,E1 -18573.293,E2 -18573.293} C_VEL
LIN {X 0,Y 256.124,Z 323.577,A -85,B 0,C 180,E1 -18577.272,E2 -18577.272} C_VEL
LIN {X 0,Y 256.085,Z 323.586,A -85,B 0,C 180,E1 -18581.305,E2 -18581.305} C_VEL
LIN {X 0,Y 256.876,Z 326.573,A -85,B 0,C 180,E1 -18582.775,E2 -18582.775} C_VEL
LIN {X 0,Y 259.301,Z 330.712,A -85,B 0,C 180,E1 -18583.387,E2 -18583.387} C_VEL
LIN {X 0,Y 266.85,Z 343.758,A -85,B 0,C 180,E1 -18585.191,E2 -18585.191} C_VEL
LIN {X 0,Y 274.512,Z 358.601,A -85,B 0,C 180,E1 -18586.925,E2 -18586.925} C_VEL
LIN {X 0,Y 279.922,Z 371.082,A -85,B 0,C 180,E1 -18588.131,E2 -18588.131} C_VEL
LIN {X 0,Y 277.306,Z 434.36,A -85,B 0,C 180,E1 -18589.77,E2 -18589.77} C_VEL
LIN {X 0,Y 276.056,Z 447.589,A -85,B 0,C 180,E1 -18590.383,E2 -18590.383} C_VEL
LIN {X 0,Y 274.451,Z 460.088,A -85,B 0,C 180,E1 -18591.259,E2 -18591.259} C_VEL
LIN {X 0,Y 272.727,Z 470.658,A -85,B 0,C 180,E1 -18592.263,E2 -18592.263} C_VEL
LIN {X 0,Y 270.617,Z 481.668,A -85,B 0,C 180,E1 -18593.619,E2 -18593.619} C_VEL
LIN {X 0,Y 268.121,Z 492.188,A -85,B 0,C 180,E1 -18595.241,E2 -18595.241} C_VEL
LIN {X 0,Y 265.498,Z 501.948,A -85,B 0,C 180,E1 -18597.135,E2 -18597.135} C_VEL
LIN {X 0,Y 263.271,Z 509.549,A -85,B 0,C 180,E1 -18598.975,E2 -18598.975} C_VEL
LIN {X 0,Y 260.767,Z 517.565,A -85,B 0,C 180,E1 -18601.419,E2 -18601.419} C_VEL
LIN {X 0,Y 258.836,Z 523.327,A -85,B 0,C 180,E1 -18603.642,E2 -18603.642} C_VEL
LIN {X 0,Y 257.347,Z 527.785,A -85,B 0,C 180,E1 -18605.817,E2 -18605.817} C_VEL
LIN {X 0,Y 256.031,Z 531.606,A -85,B 0,C 180,E1 -18608.248,E2 -18608.248} C_VEL
LIN {X 0,Y 255.079,Z 534.35,A -85,B 0,C 180,E1 -18610.692,E2 -18610.692} C_VEL
LIN {X 0,Y 254.558,Z 535.627,A -85,B 0,C 180,E1 -18612.319,E2 -18612.319} C_VEL
LIN {X 0,Y 254.24,Z 536.491,A -85,B 0,C 180,E1 -18613.952,E2 -18613.952} C_VEL
LIN {X 0,Y 254.072,Z 536.898,A -85,B 0,C 180,E1 -18615.583,E2 -18615.583} C_VEL
LIN {X 0,Y 253.896,Z 536.909,A -85,B 0,C 180,E1 -18617.205,E2 -18617.205} C_VEL
LIN {X 0,Y 253.778,Z 536.53,A -85,B 0,C 180,E1 -18618.821,E2 -18618.821} C_VEL
LIN {X 0,Y 253.785,Z 535.745,A -85,B 0,C 180,E1 -18620.435,E2 -18620.435} C_VEL
LIN {X 0,Y 253.889,Z 534.513,A -85,B 0,C 180,E1 -18622.043,E2 -18622.043} C_VEL
LIN {X 0,Y 254.19,Z 531.862,A -85,B 0,C 180,E1 -18624.478,E2 -18624.478} C_VEL
LIN {X 0,Y 254.577,Z 528.294,A -85,B 0,C 180,E1 -18626.834,E2 -18626.834} C_VEL
LIN {X 0,Y 255.168,Z 523.576,A -85,B 0,C 180,E1 -18629.21,E2 -18629.21} C_VEL
LIN {X 0,Y 256.163,Z 516.5,A -85,B 0,C 180,E1 -18631.964,E2 -18631.964} C_VEL
LIN {X 0,Y 257.538,Z 508.793,A -85,B 0,C 180,E1 -18634.303,E2 -18634.303} C_VEL
LIN {X 0,Y 258.99,Z 499.16,A -85,B 0,C 180,E1 -18636.621,E2 -18636.621} C_VEL
LIN {X 0,Y 260.529,Z 490.25,A -85,B 0,C 180,E1 -18638.336,E2 -18638.336} C_VEL
LIN {X 0,Y 262.271,Z 479.293,A -85,B 0,C 180,E1 -18640.03,E2 -18640.03} C_VEL
LIN {X 0,Y 263.73,Z 466.857,A -85,B 0,C 180,E1 -18641.528,E2 -18641.528} C_VEL
LIN {X 0,Y 264.863,Z 454.653,A -85,B 0,C 180,E1 -18642.644,E2 -18642.644} C_VEL
LIN {X 0,Y 265.815,Z 441.713,A -85,B 0,C 180,E1 -18643.472,E2 -18643.472} C_VEL
LIN {X 0,Y 266.508,Z 429.176,A -85,B 0,C 180,E1 -18643.977,E2 -18643.977} C_VEL
LIN {X 0,Y 268.506,Z 361.477,A -85,B 0,C 180,E1 -18645.746,E2 -18645.746} C_VEL
LIN {X 0,Y 267.104,Z 353.402,A -85,B 0,C 180,E1 -18646.105,E2 -18646.105} C_VEL
LIN {X 0,Y 261.303,Z 337.276,A -85,B 0,C 180,E1 -18647.127,E2 -18647.127} C_VEL
LIN {X 0,Y 256.622,Z 325.722,A -85,B 0,C 180,E1 -18647.975,E2 -18647.975} C_VEL
LIN {X 0,Y 256.142,Z 323.583,A -85,B 0,C 180,E1 -18648.911,E2 -18648.911} C_VEL
LIN {X 0,Y 256.064,Z 323.588,A -85,B 0,C 180,E1 -18652.596,E2 -18652.596} C_VEL
LIN {X 0,Y 256.067,Z 323.589,A -85,B 0,C 180,E1 -18656.047,E2 -18656.047} C_VEL
LIN {X 0,Y 256.039,Z 323.589,A -85,B 0,C 180,E1 -18659.607,E2 -18659.607} C_VEL
LIN {X 0,Y 256.064,Z 323.585,A -85,B 0,C 180,E1 -18663.292,E2 -18663.292} C_VEL
LIN {X 0,Y 256.11,Z 323.582,A -85,B 0,C 180,E1 -18667.268,E2 -18667.268} C_VEL
LIN {X 0,Y 256.015,Z 323.591,A -85,B 0,C 180,E1 -18671.209,E2 -18671.209} C_VEL
LIN {X 0,Y 256.014,Z 323.589,A -85,B 0,C 180,E1 -18675.538,E2 -18675.538} C_VEL
LIN {X 0,Y 256.014,Z 323.589,A -85,B 0,C 180,E1 -18678.788,E2 -18678.788} C_VEL
LIN {X 0,Y 256.121,Z 323.579,A -85,B 0,C 180,E1 -18682.865,E2 -18682.865} C_VEL
LIN {X 0,Y 256.06,Z 323.581,A -85,B 0,C 180,E1 -18686.706,E2 -18686.706} C_VEL
LIN {X 0,Y 256.034,Z 323.588,A -85,B 0,C 180,E1 -18690.39,E2 -18690.39} C_VEL
LIN {X 0,Y 256.06,Z 323.575,A -85,B 0,C 180,E1 -18693.95,E2 -18693.95} C_VEL
LIN {X 0,Y 256.051,Z 323.587,A -85,B 0,C 180,E1 -18697.401,E2 -18697.401} C_VEL
LIN {X 0,Y 256.098,Z 323.581,A -85,B 0,C 180,E1 -18700.773,E2 -18700.773} C_VEL
LIN {X 0,Y 256.206,Z 323.556,A -85,B 0,C 180,E1 -18704.079,E2 -18704.079} C_VEL
LIN {X 0,Y 256.262,Z 323.561,A -85,B 0,C 180,E1 -18708.932,E2 -18708.932} C_VEL
LIN {X 0,Y 256.448,Z 323.537,A -85,B 0,C 180,E1 -18712.124,E2 -18712.124} C_VEL
LIN {X 0,Y 256.447,Z 323.533,A -85,B 0,C 180,E1 -18716.858,E2 -18716.858} C_VEL
LIN {X 0,Y 256.515,Z 323.524,A -85,B 0,C 180,E1 -18717.446,E2 -18717.446} C_VEL
LIN {X 0,Y 255.961,Z 323.599,A -85,B 0,C 180,E1 -18718.758,E2 -18718.758} C_VEL
LIN {X 0,Y 254.386,Z 323.796,A -85,B 0,C 180,E1 -18720.046,E2 -18720.046} C_VEL
LIN {X 0,Y 250.511,Z 324.276,A -85,B 0,C 180,E1 -18722.634,E2 -18722.634} C_VEL
LIN {X 0,Y 249.377,Z 324.415,A -85,B 0,C 180,E1 -18723.986,E2 -18723.986} C_VEL
LIN {X 0,Y 249.271,Z 324.42,A -85,B 0,C 180,E1 -18724.446,E2 -18724.446} C_VEL
LIN {X 0,Y 249.428,Z 324.408,A -85,B 0,C 180,E1 -18728.099,E2 -18728.099} C_VEL
LIN {X 0,Y 249.179,Z 324.441,A -85,B 0,C 180,E1 -18733.04,E2 -18733.04} C_VEL
LIN {X 0,Y 249.166,Z 324.435,A -85,B 0,C 180,E1 -18736.468,E2 -18736.468} C_VEL
LIN {X 0,Y 249.074,Z 324.456,A -85,B 0,C 180,E1 -18741.519,E2 -18741.519} C_VEL
LIN {X 0,Y 249.106,Z 324.455,A -85,B 0,C 180,E1 -18745.474,E2 -18745.474} C_VEL
LIN {X 0,Y 249.057,Z 324.457,A -85,B 0,C 180,E1 -18748.986,E2 -18748.986} C_VEL
LIN {X 0,Y 249.024,Z 324.461,A -85,B 0,C 180,E1 -18752.427,E2 -18752.427} C_VEL
LIN {X 0,Y 249.021,Z 324.462,A -85,B 0,C 180,E1 -18756.347,E2 -18756.347} C_VEL
LIN {X 0,Y 248.984,Z 324.466,A -85,B 0,C 180,E1 -18760.482,E2 -18760.482} C_VEL
LIN {X 0,Y 248.988,Z 324.469,A -85,B 0,C 180,E1 -18764.883,E2 -18764.883} C_VEL
LIN {X 0,Y 249.012,Z 324.467,A -85,B 0,C 180,E1 -18767.364,E2 -18767.364} C_VEL
LIN {X 0,Y 249.044,Z 324.464,A -85,B 0,C 180,E1 -18772.2,E2 -18772.2} C_VEL
LIN {X 0,Y 249.1,Z 324.662,A -85,B 0,C 180,E1 -18775.377,E2 -18775.377} C_VEL
LIN {X 0,Y 251.654,Z 336.269,A -85,B 0,C 180,E1 -18779.824,E2 -18779.824} C_VEL
LIN {X 0,Y 252.012,Z 338.35,A -85,B 0,C 180,E1 -18780.585,E2 -18780.585} C_VEL
LIN {X 0,Y 257.012,Z 352.422,A -85,B 0,C 180,E1 -18781.537,E2 -18781.537} C_VEL
LIN {X 0,Y 261.269,Z 385.419,A -85,B 0,C 180,E1 -18782.925,E2 -18782.925} C_VEL
LIN {X 0,Y 259.624,Z 447.68,A -85,B 0,C 180,E1 -18784.658,E2 -18784.658} C_VEL
LIN {X 0,Y 258.628,Z 461.458,A -85,B 0,C 180,E1 -18785.359,E2 -18785.359} C_VEL
LIN {X 0,Y 257.382,Z 473.291,A -85,B 0,C 180,E1 -18786.251,E2 -18786.251} C_VEL
LIN {X 0,Y 255.995,Z 484.507,A -85,B 0,C 180,E1 -18787.398,E2 -18787.398} C_VEL
LIN {X 0,Y 254.186,Z 496.15,A -85,B 0,C 180,E1 -18788.936,E2 -18788.936} C_VEL
LIN {X 0,Y 252.713,Z 505.564,A -85,B 0,C 180,E1 -18790.507,E2 -18790.507} C_VEL
LIN {X 0,Y 251.259,Z 515.226,A -85,B 0,C 180,E1 -18792.502,E2 -18792.502} C_VEL
LIN {X 0,Y 249.911,Z 523.105,A -85,B 0,C 180,E1 -18794.506,E2 -18794.506} C_VEL
LIN {X 0,Y 248.569,Z 530.779,A -85,B 0,C 180,E1 -18796.928,E2 -18796.928} C_VEL
